DECL E6POS XP382={x 2180.9021,y 585.806824,z 1369.54504,a -78.3736267,b 58.1377296,c -93.7700119,s 6,t 27,e1 0.0,e2 0.0,e3 0.0,e4 0.0,e5 0.0,e6 0.0}
DECL FDAT FP382={TOOL_NO 1,BASE_NO 0,IPO_FRAME #BASE}
DECL PDAT PPDAT276={VEL 100.0,ACC 100.0,APO_DIST 100.0}
DECL E6POS XP383={x 1882.12,y 578.306091,z 982.650513,a -78.3796005,b 58.1366501,c -93.7758102,s 6,t 27,e1 0.0,e2 0.0,e3 0.0,e4 0.0,e5 0.0,e6 0.0}
DECL FDAT FP383={TOOL_NO 1,BASE_NO 0,IPO_FRAME #BASE}
DECL PDAT PPDAT277={VEL 100.0,ACC 100.0,APO_DIST 100.0}
DECL E6POS XP384={x 1882.09204,y 578.297729,z 939.258484,a -78.3842316,b 58.1358299,c -93.7813263,s 6,t 27,e1 0.0,e2 0.0,e3 0.0,e4 0.0,e5 0.0,e6 0.0}
DECL FDAT FP384={TOOL_NO 1,BASE_NO 0,IPO_FRAME #BASE}
DECL PDAT PPDAT278={VEL 100.0,ACC 100.0,APO_DIST 100.0}
DECL E6POS XP385={x 1882.10596,y 497.070801,z 1745.22595,a -88.2604828,b 58.8505211,c -105.352699,s 6,t 19,e1 0.0,e2 0.0,e3 0.0,e4 0.0,e5 0.0,e6 0.0}
DECL FDAT FP385={TOOL_NO 1,BASE_NO 0,IPO_FRAME #BASE}
DECL PDAT PPDAT279={VEL 100.0,ACC 100.0,APO_DIST 100.0}
DECL E6POS XP386={x 1882.10498,y 109.2248,z 1745.24194,a -43.191761,b 40.938839,c -48.9825897,s 6,t 19,e1 0.0,e2 0.0,e3 0.0,e4 0.0,e5 0.0,e6 0.0}
DECL FDAT FP386={TOOL_NO 1,BASE_NO 0,IPO_FRAME #BASE}
DECL PDAT PPDAT280={VEL 100.0,ACC 100.0,APO_DIST 100.0}
DECL E6POS XP387={x 1882.12097,y 109.308701,z 1745.27405,a 7.98916388,b -56.2097092,c 176.517807,s 6,t 27,e1 0.0,e2 0.0,e3 0.0,e4 0.0,e5 0.0,e6 0.0}
DECL FDAT FP387={TOOL_NO 1,BASE_NO 0,IPO_FRAME #BASE}
DECL PDAT PPDAT281={VEL 100.0,ACC 100.0,APO_DIST 100.0}
DECL E6POS XP388={x 1580.30603,y 109.311897,z 1338.53003,a 29.1239491,b -3.817909,c -177.125595,s 6,t 27,e1 0.0,e2 0.0,e3 0.0,e4 0.0,e5 0.0,e6 0.0}
DECL FDAT FP388={TOOL_NO 1,BASE_NO 0,IPO_FRAME #BASE}
DECL PDAT PPDAT282={VEL 100.0,ACC 100.0,APO_DIST 100.0}
DECL E6POS XP389={x 55.3110695,y 943.681396,z 1978.17395,a -6.70130014,b 52.5186882,c -94.4837189,s 2,t 11,e1 0.0,e2 0.0,e3 0.0,e4 0.0,e5 0.0,e6 0.0}
DECL FDAT FP389={TOOL_NO 1,BASE_NO 0,IPO_FRAME #BASE}
DECL PDAT PPDAT283={VEL 100.0,ACC 25.0,APO_DIST 100.0}
DECL E6POS XP390={x 1620.0,y 0.0,z 2195.0,a -90.0,b 59.9998817,c -90.0,s 2,t 2,e1 0.0,e2 0.0,e3 0.0,e4 0.0,e5 0.0,e6 0.0}
DECL FDAT FP390={TOOL_NO 1,BASE_NO 0,IPO_FRAME #BASE}
DECL PDAT PPDAT284={VEL 100.0,ACC 100.0,APO_DIST 100.0}
DECL E6POS XP391={x 1721.71704,y 98.0797729,z 1269.401,a -89.9984894,b 59.9988289,c -89.9980927,s 6,t 27,e1 0.0,e2 0.0,e3 0.0,e4 0.0,e5 0.0,e6 0.0}
DECL FDAT FP391={TOOL_NO 1,BASE_NO 0,IPO_FRAME #BASE}
DECL PDAT PPDAT285={VEL 100.0,ACC 100.0,APO_DIST 100.0}
DECL E6POS XP392={x 1730.89404,y 101.730797,z 1269.375,a -89.9981079,b 59.9989815,c -89.9963837,s 6,t 27,e1 0.0,e2 0.0,e3 0.0,e4 0.0,e5 0.0,e6 0.0}
DECL FDAT FP392={TOOL_NO 1,BASE_NO 0,IPO_FRAME #BASE}
DECL PDAT PPDAT286={VEL 100.0,ACC 100.0,APO_DIST 100.0}
DECL E6POS XP393={x 1730.89404,y 101.730797,z 1269.375,a -89.9981079,b 59.9989815,c -89.9963837,s 6,t 27,e1 0.0,e2 0.0,e3 0.0,e4 0.0,e5 0.0,e6 0.0}
DECL FDAT FP393={TOOL_NO 1,BASE_NO 0,IPO_FRAME #BASE}
DECL LDAT LCPDAT97={VEL 2.0,ACC 100.0,APO_DIST 100.0,APO_FAC 50.0}
DECL E6POS XP394={x 1730.89404,y 101.730797,z 1269.375,a -89.9981079,b 59.9989815,c -89.9963837,s 6,t 27,e1 0.0,e2 0.0,e3 0.0,e4 0.0,e5 0.0,e6 0.0}
DECL FDAT FP394={TOOL_NO 1,BASE_NO 0,IPO_FRAME #BASE}
DECL LDAT LCPDAT98={VEL 2.0,ACC 100.0,APO_DIST 100.0,APO_FAC 50.0}
DECL E6POS XP395={x 1721.30396,y 101.718201,z 1269.37402,a -89.9990005,b 59.9981804,c -89.9970932,s 6,t 27,e1 0.0,e2 0.0,e3 0.0,e4 0.0,e5 0.0,e6 0.0}
DECL FDAT FP395={TOOL_NO 1,BASE_NO 0,IPO_FRAME #BASE}
DECL LDAT LCPDAT99={VEL 2.0,ACC 100.0,APO_DIST 100.0,APO_FAC 50.0}
DECL E6POS XP396={x 1721.30896,y 95.7696762,z 1269.37903,a -89.9983902,b 59.9984283,c -89.9962692,s 6,t 27,e1 0.0,e2 0.0,e3 0.0,e4 0.0,e5 0.0,e6 0.0}
DECL FDAT FP396={TOOL_NO 1,BASE_NO 0,IPO_FRAME #BASE}
DECL LDAT LCPDAT100={VEL 2.0,ACC 100.0,APO_DIST 100.0,APO_FAC 50.0}
DECL E6POS XP397={x 1727.48706,y 95.7749023,z 1269.40405,a -89.994957,b 59.999321,c -89.9919434,s 6,t 27,e1 0.0,e2 0.0,e3 0.0,e4 0.0,e5 0.0,e6 0.0}
DECL FDAT FP397={TOOL_NO 1,BASE_NO 0,IPO_FRAME #BASE}
DECL LDAT LCPDAT101={VEL 2.0,ACC 100.0,APO_DIST 100.0,APO_FAC 50.0}
DECL E6POS XP398={x 1727.49194,y 99.8509369,z 1269.41504,a -89.9935379,b 60.0002289,c -89.9901505,s 6,t 27,e1 0.0,e2 0.0,e3 0.0,e4 0.0,e5 0.0,e6 0.0}
DECL FDAT FP398={TOOL_NO 1,BASE_NO 0,IPO_FRAME #BASE}
DECL LDAT LCPDAT102={VEL 2.0,ACC 100.0,APO_DIST 100.0,APO_FAC 50.0}
DECL E6POS XP399={x 1727.49194,y 99.8509369,z 1269.41504,a -89.9935379,b 60.0002289,c -89.9901505,s 6,t 27,e1 0.0,e2 0.0,e3 0.0,e4 0.0,e5 0.0,e6 0.0}
DECL FDAT FP399={TOOL_NO 1,BASE_NO 0,IPO_FRAME #BASE}
DECL PDAT PPDAT287={VEL 100.0,ACC 100.0,APO_DIST 100.0}
DECL E6POS XP400={x 1727.49805,y 9.73986816,z 1288.27502,a -89.9890137,b 68.490097,c -89.9850311,s 6,t 27,e1 0.0,e2 0.0,e3 0.0,e4 0.0,e5 0.0,e6 0.0}
DECL FDAT FP400={TOOL_NO 1,BASE_NO 0,IPO_FRAME #BASE}
DECL PDAT PPDAT288={VEL 100.0,ACC 100.0,APO_DIST 100.0}
DECL E6POS XP401={x 1825.16003,y 8.47059917,z 1266.86694,a -89.9738693,b 68.4893494,c -89.9686432,s 6,t 27,e1 0.0,e2 0.0,e3 0.0,e4 0.0,e5 0.0,e6 0.0}
DECL FDAT FP401={TOOL_NO 1,BASE_NO 0,IPO_FRAME #BASE}
DECL PDAT PPDAT289={VEL 100.0,ACC 100.0,APO_DIST 100.0}
DECL E6POS XP402={x 1825.16003,y 8.47059917,z 1266.86694,a -89.9738693,b 68.4893494,c -89.9686432,s 6,t 27,e1 0.0,e2 0.0,e3 0.0,e4 0.0,e5 0.0,e6 0.0}
DECL FDAT FP402={TOOL_NO 1,BASE_NO 0,IPO_FRAME #BASE}
DECL LDAT LCPDAT103={VEL 2.0,ACC 100.0,APO_DIST 100.0,APO_FAC 50.0}
DECL E6POS XP403={x 1795.98206,y 8.45187664,z 1267.44702,a -89.9924164,b 68.4888229,c -89.9880981,s 6,t 27,e1 0.0,e2 0.0,e3 0.0,e4 0.0,e5 0.0,e6 0.0}
DECL FDAT FP403={TOOL_NO 1,BASE_NO 0,IPO_FRAME #BASE}
DECL LDAT LCPDAT104={VEL 2.0,ACC 100.0,APO_DIST 100.0,APO_FAC 50.0}
DECL E6POS XP404={x 1762.83203,y 8.4597578,z 1218.80896,a -89.9986496,b 68.4880295,c -89.995163,s 6,t 27,e1 0.0,e2 0.0,e3 0.0,e4 0.0,e5 0.0,e6 0.0}
DECL FDAT FP404={TOOL_NO 1,BASE_NO 0,IPO_FRAME #BASE}
DECL LDAT LCPDAT105={VEL 2.0,ACC 100.0,APO_DIST 100.0,APO_FAC 50.0}
DECL E6POS XP405={x 1714.34094,y 9.04022121,z 1220.41504,a -90.0047531,b 68.486908,c -90.0016937,s 6,t 27,e1 0.0,e2 0.0,e3 0.0,e4 0.0,e5 0.0,e6 0.0}
DECL FDAT FP405={TOOL_NO 1,BASE_NO 0,IPO_FRAME #BASE}
DECL LDAT LCPDAT106={VEL 2.0,ACC 100.0,APO_DIST 100.0,APO_FAC 50.0}
DECL E6POS XP406={x 1787.46497,y 1.54117298,z 1305.14099,a -89.9851837,b 68.4879913,c -89.9798126,s 6,t 27,e1 0.0,e2 0.0,e3 0.0,e4 0.0,e5 0.0,e6 0.0}
DECL FDAT FP406={TOOL_NO 1,BASE_NO 0,IPO_FRAME #BASE}
DECL PDAT PPDAT290={VEL 100.0,ACC 100.0,APO_DIST 100.0}
DECL E6POS XP407={x 6.87235498,y -107.955902,z 3197.98999,a -95.3498535,b 3.01419806,c -0.477443188,s 2,t 10,e1 0.0,e2 0.0,e3 0.0,e4 0.0,e5 0.0,e6 0.0}
DECL FDAT FP407={TOOL_NO 1,BASE_NO 0,IPO_FRAME #BASE}
DECL PDAT PPDAT291={VEL 100.0,ACC 100.0,APO_DIST 100.0}
DECL E6POS XP408={x -2321.86401,y -437.479095,z 1523.60596,a -44.4752808,b -52.6538696,c 48.7558517,s 6,t 26,e1 0.0,e2 0.0,e3 0.0,e4 0.0,e5 0.0,e6 0.0}
DECL FDAT FP408={TOOL_NO 1,BASE_NO 0,IPO_FRAME #BASE}
DECL PDAT PPDAT292={VEL 100.0,ACC 100.0,APO_DIST 100.0}
DECL E6POS XP409={x 2083.62109,y -1113.97803,z 1523.60205,a 96.7235031,b -52.6538696,c 48.7562599,s 6,t 26,e1 0.0,e2 0.0,e3 0.0,e4 0.0,e5 0.0,e6 0.0}
DECL FDAT FP409={TOOL_NO 1,BASE_NO 0,IPO_FRAME #BASE}
DECL PDAT PPDAT293={VEL 100.0,ACC 100.0,APO_DIST 100.0}
DECL E6POS XP410={x 1843.23206,y -297.672211,z 1892.20703,a -104.636902,b 62.3937492,c -97.5844193,s 6,t 18,e1 0.0,e2 0.0,e3 0.0,e4 0.0,e5 0.0,e6 0.0}
DECL FDAT FP410={TOOL_NO 1,BASE_NO 0,IPO_FRAME #BASE}
DECL PDAT PPDAT294={VEL 100.0,ACC 100.0,APO_DIST 100.0}
DECL E6POS XP411={x 1891.35901,y -309.263092,z 920.833923,a -96.7764893,b 62.3960686,c -97.579422,s 6,t 18,e1 0.0,e2 0.0,e3 0.0,e4 0.0,e5 0.0,e6 0.0}
DECL FDAT FP411={TOOL_NO 1,BASE_NO 0,IPO_FRAME #BASE}
DECL PDAT PPDAT295={VEL 100.0,ACC 100.0,APO_DIST 100.0}
DECL E6POS XP412={x 1891.36206,y -309.26709,z 1131.79297,a -96.7787933,b 62.396759,c -97.5819702,s 6,t 18,e1 0.0,e2 0.0,e3 0.0,e4 0.0,e5 0.0,e6 0.0}
DECL FDAT FP412={TOOL_NO 1,BASE_NO 0,IPO_FRAME #BASE}
DECL PDAT PPDAT296={VEL 100.0,ACC 100.0,APO_DIST 100.0}
DECL E6POS XP413={x 1891.35803,y -150.701401,z 1131.78699,a -96.7800903,b 62.3966904,c -97.5833969,s 6,t 18,e1 0.0,e2 0.0,e3 0.0,e4 0.0,e5 0.0,e6 0.0}
DECL FDAT FP413={TOOL_NO 1,BASE_NO 0,IPO_FRAME #BASE}
DECL PDAT PPDAT297={VEL 100.0,ACC 100.0,APO_DIST 100.0}
DECL E6POS XP414={x 1891.39001,y -150.693405,z 1087.95801,a -96.7599106,b 62.3970795,c -97.5624237,s 6,t 18,e1 0.0,e2 0.0,e3 0.0,e4 0.0,e5 0.0,e6 0.0}
DECL FDAT FP414={TOOL_NO 1,BASE_NO 0,IPO_FRAME #BASE}
DECL PDAT PPDAT298={VEL 100.0,ACC 100.0,APO_DIST 100.0}
DECL E6POS XP415={x 1788.51697,y 1.54148304,z 1085.06396,a -89.9759216,b 68.4883728,c -89.9696884,s 6,t 27,e1 0.0,e2 0.0,e3 0.0,e4 0.0,e5 0.0,e6 0.0}
DECL FDAT FP415={TOOL_NO 1,BASE_NO 0,IPO_FRAME #BASE}
DECL PDAT PPDAT299={VEL 100.0,ACC 100.0,APO_DIST 100.0}
DECL E6POS XP416={x 1788.51697,y 1.54148304,z 1085.06396,a -89.9759216,b 68.4883728,c -89.9696884,s 6,t 27,e1 0.0,e2 0.0,e3 0.0,e4 0.0,e5 0.0,e6 0.0}
DECL FDAT FP416={TOOL_NO 1,BASE_NO 0,IPO_FRAME #BASE}
DECL LDAT LCPDAT107={VEL 2.0,ACC 100.0,APO_DIST 100.0,APO_FAC 50.0}
DECL E6POS XP417={x 1781.58704,y -240.441803,z 1083.771,a -89.9750977,b 68.4889297,c -89.9688263,s 6,t 18,e1 0.0,e2 0.0,e3 0.0,e4 0.0,e5 0.0,e6 0.0}
DECL FDAT FP417={TOOL_NO 1,BASE_NO 0,IPO_FRAME #BASE}
DECL LDAT LCPDAT108={VEL 2.0,ACC 100.0,APO_DIST 100.0,APO_FAC 50.0}
DECL E6POS XP418={x 1857.57495,y -189.287598,z 1190.64795,a -5.03419781,b 68.481781,c -89.9884262,s 6,t 50,e1 0.0,e2 0.0,e3 0.0,e4 0.0,e5 0.0,e6 0.0}
DECL FDAT FP418={TOOL_NO 1,BASE_NO 0,IPO_FRAME #BASE}
DECL PDAT PPDAT300={VEL 100.0,ACC 100.0,APO_DIST 100.0}
DECL E6POS XP419={x 1857.57104,y -189.290497,z 1089.01599,a -5.03386116,b 68.4827805,c -89.9877167,s 6,t 50,e1 0.0,e2 0.0,e3 0.0,e4 0.0,e5 0.0,e6 0.0}
DECL FDAT FP419={TOOL_NO 1,BASE_NO 0,IPO_FRAME #BASE}
DECL PDAT PPDAT301={VEL 100.0,ACC 100.0,APO_DIST 100.0}
DECL E6POS XP420={x 1857.57104,y -189.290497,z 1089.01599,a -5.03386116,b 68.4827805,c -89.9877167,s 6,t 50,e1 0.0,e2 0.0,e3 0.0,e4 0.0,e5 0.0,e6 0.0}
DECL FDAT FP420={TOOL_NO 1,BASE_NO 0,IPO_FRAME #BASE}
DECL LDAT LCPDAT109={VEL 2.0,ACC 100.0,APO_DIST 100.0,APO_FAC 50.0}
DECL E6POS XP421={x 2014.16101,y -191.725006,z 1089.02905,a -5.03730679,b 68.4811783,c -89.9894867,s 6,t 50,e1 0.0,e2 0.0,e3 0.0,e4 0.0,e5 0.0,e6 0.0}
DECL FDAT FP421={TOOL_NO 1,BASE_NO 0,IPO_FRAME #BASE}
DECL LDAT LCPDAT110={VEL 2.0,ACC 100.0,APO_DIST 100.0,APO_FAC 50.0}
DECL E6POS XP422={x 2014.16101,y -191.725006,z 1089.02905,a -5.03730679,b 68.4811783,c -89.9894867,s 6,t 50,e1 0.0,e2 0.0,e3 0.0,e4 0.0,e5 0.0,e6 0.0}
DECL FDAT FP422={TOOL_NO 1,BASE_NO 0,IPO_FRAME #BASE}
DECL PDAT PPDAT302={VEL 100.0,ACC 100.0,APO_DIST 100.0}
DECL E6POS XP423={x 1938.26904,y -244.236496,z 1088.59204,a -91.4427872,b 68.4859772,c -89.9945831,s 6,t 18,e1 0.0,e2 0.0,e3 0.0,e4 0.0,e5 0.0,e6 0.0}
DECL FDAT FP423={TOOL_NO 1,BASE_NO 0,IPO_FRAME #BASE}
DECL PDAT PPDAT303={VEL 100.0,ACC 100.0,APO_DIST 100.0}
DECL E6POS XP424={x 1938.27197,y -244.231201,z 1081.43005,a -91.440033,b 68.4871368,c -89.9929428,s 6,t 18,e1 0.0,e2 0.0,e3 0.0,e4 0.0,e5 0.0,e6 0.0}
DECL FDAT FP424={TOOL_NO 1,BASE_NO 0,IPO_FRAME #BASE}
DECL PDAT PPDAT304={VEL 100.0,ACC 100.0,APO_DIST 100.0}
DECL E6POS XP425={x 1938.27197,y -244.231201,z 1081.43005,a -91.440033,b 68.4871368,c -89.9929428,s 6,t 18,e1 0.0,e2 0.0,e3 0.0,e4 0.0,e5 0.0,e6 0.0}
DECL FDAT FP425={TOOL_NO 1,BASE_NO 0,IPO_FRAME #BASE}
DECL LDAT LCPDAT111={VEL 2.0,ACC 100.0,APO_DIST 100.0,APO_FAC 50.0}
DECL E6POS XP426={x 1951.03503,y 280.272705,z 1084.44604,a -91.4313889,b 68.4940109,c -89.9844894,s 6,t 27,e1 0.0,e2 0.0,e3 0.0,e4 0.0,e5 0.0,e6 0.0}
DECL FDAT FP426={TOOL_NO 1,BASE_NO 0,IPO_FRAME #BASE}
DECL LDAT LCPDAT112={VEL 2.0,ACC 100.0,APO_DIST 100.0,APO_FAC 50.0}
DECL E6POS XP427={x 1951.03503,y 280.272705,z 1084.44604,a -91.4313889,b 68.4940109,c -89.9844894,s 6,t 27,e1 0.0,e2 0.0,e3 0.0,e4 0.0,e5 0.0,e6 0.0}
DECL FDAT FP427={TOOL_NO 1,BASE_NO 0,IPO_FRAME #BASE}
DECL PDAT PPDAT305={VEL 100.0,ACC 100.0,APO_DIST 100.0}
DECL E6POS XP428={x 2026.85901,y 334.200104,z 1105.98096,a -4.45665598,b 68.4910431,c -89.9797287,s 6,t 51,e1 0.0,e2 0.0,e3 0.0,e4 0.0,e5 0.0,e6 0.0}
DECL FDAT FP428={TOOL_NO 1,BASE_NO 0,IPO_FRAME #BASE}
DECL PDAT PPDAT306={VEL 100.0,ACC 100.0,APO_DIST 100.0}
DECL E6POS XP429={x 2026.85596,y 334.200012,z 1089.23096,a -4.45706797,b 68.4920731,c -89.9801331,s 6,t 51,e1 0.0,e2 0.0,e3 0.0,e4 0.0,e5 0.0,e6 0.0}
DECL FDAT FP429={TOOL_NO 1,BASE_NO 0,IPO_FRAME #BASE}
DECL LDAT LCPDAT113={VEL 2.0,ACC 100.0,APO_DIST 100.0,APO_FAC 50.0}
DECL E6POS XP430={x 2026.85596,y 334.200012,z 1089.23096,a -4.45706797,b 68.4920731,c -89.9801331,s 6,t 51,e1 0.0,e2 0.0,e3 0.0,e4 0.0,e5 0.0,e6 0.0}
DECL FDAT FP430={TOOL_NO 1,BASE_NO 0,IPO_FRAME #BASE}
DECL LDAT LCPDAT114={VEL 2.0,ACC 100.0,APO_DIST 100.0,APO_FAC 50.0}
DECL E6POS XP431={x 1867.99402,y 335.831604,z 1091.06995,a -4.45940113,b 68.4928665,c -89.9819336,s 6,t 51,e1 0.0,e2 0.0,e3 0.0,e4 0.0,e5 0.0,e6 0.0}
DECL FDAT FP431={TOOL_NO 1,BASE_NO 0,IPO_FRAME #BASE}
DECL LDAT LCPDAT115={VEL 2.0,ACC 100.0,APO_DIST 100.0,APO_FAC 50.0}
DECL E6POS XP432={x 1867.99402,y 335.831604,z 1091.06995,a -4.45940113,b 68.4928665,c -89.9819336,s 6,t 51,e1 0.0,e2 0.0,e3 0.0,e4 0.0,e5 0.0,e6 0.0}
DECL FDAT FP432={TOOL_NO 1,BASE_NO 0,IPO_FRAME #BASE}
DECL PDAT PPDAT307={VEL 100.0,ACC 100.0,APO_DIST 100.0}
DECL E6POS XP433={x 1801.823,y 283.612,z 1101.84595,a -95.9969177,b 68.3930435,c -93.1611633,s 6,t 27,e1 0.0,e2 0.0,e3 0.0,e4 0.0,e5 0.0,e6 0.0}
DECL FDAT FP433={TOOL_NO 1,BASE_NO 0,IPO_FRAME #BASE}
DECL PDAT PPDAT308={VEL 100.0,ACC 100.0,APO_DIST 100.0}
DECL E6POS XP434={x 1801.83801,y 283.613007,z 1086.224,a -95.9930725,b 68.3924332,c -93.1558304,s 6,t 27,e1 0.0,e2 0.0,e3 0.0,e4 0.0,e5 0.0,e6 0.0}
DECL FDAT FP434={TOOL_NO 1,BASE_NO 0,IPO_FRAME #BASE}
DECL PDAT PPDAT309={VEL 100.0,ACC 100.0,APO_DIST 100.0}
DECL E6POS XP435={x 1801.84705,y 284.174896,z 1086.23096,a -95.9924088,b 68.3929901,c -93.1550217,s 6,t 27,e1 0.0,e2 0.0,e3 0.0,e4 0.0,e5 0.0,e6 0.0}
DECL FDAT FP435={TOOL_NO 1,BASE_NO 0,IPO_FRAME #BASE}
DECL LDAT LCPDAT116={VEL 2.0,ACC 100.0,APO_DIST 100.0,APO_FAC 50.0}
DECL E6POS XP436={x 1800.22595,y 216.311996,z 1086.229,a -95.9936371,b 68.3931732,c -93.155899,s 6,t 27,e1 0.0,e2 0.0,e3 0.0,e4 0.0,e5 0.0,e6 0.0}
DECL FDAT FP436={TOOL_NO 1,BASE_NO 0,IPO_FRAME #BASE}
DECL LDAT LCPDAT117={VEL 2.0,ACC 100.0,APO_DIST 100.0,APO_FAC 50.0}
DECL E6POS XP437={x 1800.22205,y 198.541901,z 1134.521,a -95.9973221,b 68.3924637,c -93.1600571,s 6,t 27,e1 0.0,e2 0.0,e3 0.0,e4 0.0,e5 0.0,e6 0.0}
DECL E6POS XP438={x 1800.23499,y 178.785706,z 1109.75195,a -95.9939728,b 68.3902435,c -93.1574936,s 6,t 27,e1 0.0,e2 0.0,e3 0.0,e4 0.0,e5 0.0,e6 0.0}
DECL FDAT FP438={TOOL_NO 1,BASE_NO 0,IPO_FRAME #BASE}
DECL LDAT LCPDAT118={VEL 2.0,ACC 100.0,APO_DIST 100.0,APO_FAC 50.0}
DECL E6POS XP439={x 1800.23596,y 178.768494,z 1086.354,a -95.9938278,b 68.3870468,c -93.1533966,s 6,t 27,e1 0.0,e2 0.0,e3 0.0,e4 0.0,e5 0.0,e6 0.0}
DECL FDAT FP439={TOOL_NO 1,BASE_NO 0,IPO_FRAME #BASE}
DECL LDAT LCPDAT119={VEL 2.0,ACC 100.0,APO_DIST 100.0,APO_FAC 50.0}
DECL E6POS XP440={x 1797.48499,y 99.9996567,z 1086.354,a -95.9934998,b 68.3869934,c -93.1527481,s 6,t 27,e1 0.0,e2 0.0,e3 0.0,e4 0.0,e5 0.0,e6 0.0}
DECL FDAT FP440={TOOL_NO 1,BASE_NO 0,IPO_FRAME #BASE}
DECL LDAT LCPDAT120={VEL 2.0,ACC 100.0,APO_DIST 100.0,APO_FAC 50.0}
DECL E6POS XP441={x 1708.21704,y 230.690506,z 1194.828,a -77.1536865,b 58.7134018,c -71.4141769,s 6,t 27,e1 0.0,e2 0.0,e3 0.0,e4 0.0,e5 0.0,e6 0.0}
DECL FDAT FP441={TOOL_NO 1,BASE_NO 0,IPO_FRAME #BASE}
DECL PDAT PPDAT310={VEL 100.0,ACC 100.0,APO_DIST 100.0}
DECL E6POS XP442={x 1709.53699,y 242.714905,z 1080.94397,a -77.1506729,b 58.7134705,c -71.4099426,s 6,t 27,e1 0.0,e2 0.0,e3 0.0,e4 0.0,e5 0.0,e6 0.0}
DECL FDAT FP442={TOOL_NO 1,BASE_NO 0,IPO_FRAME #BASE}
DECL PDAT PPDAT311={VEL 100.0,ACC 100.0,APO_DIST 100.0}
DECL E6POS XP443={x 1709.53699,y 242.714905,z 1080.94397,a -77.1506729,b 58.7134705,c -71.4099426,s 6,t 27,e1 0.0,e2 0.0,e3 0.0,e4 0.0,e5 0.0,e6 0.0}
DECL FDAT FP443={TOOL_NO 1,BASE_NO 0,IPO_FRAME #BASE}
DECL LDAT LCPDAT121={VEL 2.0,ACC 100.0,APO_DIST 100.0,APO_FAC 50.0}
DECL E6POS XP444={x 1706.01196,y 92.4064713,z 1079.61096,a -77.1516113,b 58.7126198,c -71.4103317,s 6,t 27,e1 0.0,e2 0.0,e3 0.0,e4 0.0,e5 0.0,e6 0.0}
DECL FDAT FP444={TOOL_NO 1,BASE_NO 0,IPO_FRAME #BASE}
DECL LDAT LCPDAT122={VEL 2.0,ACC 100.0,APO_DIST 100.0,APO_FAC 50.0}
DECL E6POS XP445={x 1706.01099,y 92.4069672,z 1289.64502,a -77.1514664,b 58.712719,c -71.4103165,s 6,t 27,e1 0.0,e2 0.0,e3 0.0,e4 0.0,e5 0.0,e6 0.0}
DECL FDAT FP445={TOOL_NO 1,BASE_NO 0,IPO_FRAME #BASE}
DECL PDAT PPDAT312={VEL 100.0,ACC 100.0,APO_DIST 100.0}
DECL E6POS XP446={x 1625.10095,y -190.573196,z 915.192627,a -77.1490631,b 58.7168884,c -71.4077988,s 6,t 18,e1 0.0,e2 0.0,e3 0.0,e4 0.0,e5 0.0,e6 0.0}
DECL FDAT FP446={TOOL_NO 1,BASE_NO 0,IPO_FRAME #BASE}
DECL PDAT PPDAT313={VEL 100.0,ACC 100.0,APO_DIST 100.0}
DECL E6POS XP447={x 1625.10095,y -190.573196,z 915.192627,a -77.1490631,b 58.7168884,c -71.4077988,s 6,t 18,e1 0.0,e2 0.0,e3 0.0,e4 0.0,e5 0.0,e6 0.0}
DECL FDAT FP447={TOOL_NO 1,BASE_NO 0,IPO_FRAME #BASE}
DECL LDAT LCPDAT123={VEL 2.0,ACC 100.0,APO_DIST 100.0,APO_FAC 50.0}
DECL E6POS XP448={x 1620.70203,y -356.353699,z 913.115417,a -77.1501923,b 58.7190208,c -71.4090805,s 6,t 18,e1 0.0,e2 0.0,e3 0.0,e4 0.0,e5 0.0,e6 0.0}
DECL FDAT FP448={TOOL_NO 1,BASE_NO 0,IPO_FRAME #BASE}
DECL LDAT LCPDAT124={VEL 2.0,ACC 100.0,APO_DIST 100.0,APO_FAC 50.0}
DECL E6POS XP449={x 1626.60706,y -375.643707,z 913.122986,a -77.1490707,b 58.7185707,c -71.40802,s 6,t 18,e1 0.0,e2 0.0,e3 0.0,e4 0.0,e5 0.0,e6 0.0}
DECL E6POS XP450={x 1651.60303,y -391.266998,z 912.728394,a -77.1474991,b 58.717701,c -71.4053802,s 6,t 18,e1 0.0,e2 0.0,e3 0.0,e4 0.0,e5 0.0,e6 0.0}
DECL FDAT FP450={TOOL_NO 1,BASE_NO 0,IPO_FRAME #BASE}
DECL LDAT LCPDAT125={VEL 2.0,ACC 100.0,APO_DIST 100.0,APO_FAC 50.0}
DECL E6POS XP451={x 1651.60303,y -391.266998,z 912.728394,a -77.1474991,b 58.717701,c -71.4053802,s 6,t 18,e1 0.0,e2 0.0,e3 0.0,e4 0.0,e5 0.0,e6 0.0}
DECL FDAT FP451={TOOL_NO 1,BASE_NO 0,IPO_FRAME #BASE}
DECL LDAT LCPDAT126={VEL 2.0,ACC 100.0,APO_DIST 100.0,APO_FAC 50.0}
DECL E6POS XP452={x 1877.198,y -398.11499,z 910.503418,a -77.1458435,b 58.7178192,c -71.4037476,s 6,t 18,e1 0.0,e2 0.0,e3 0.0,e4 0.0,e5 0.0,e6 0.0}
DECL FDAT FP452={TOOL_NO 1,BASE_NO 0,IPO_FRAME #BASE}
DECL LDAT LCPDAT127={VEL 2.0,ACC 100.0,APO_DIST 100.0,APO_FAC 50.0}
DECL E6POS XP453={x 1902.11096,y -390.78891,z 910.030579,a -77.1470032,b 58.7169991,c -71.404808,s 6,t 18,e1 0.0,e2 0.0,e3 0.0,e4 0.0,e5 0.0,e6 0.0}
DECL E6POS XP454={x 1917.34802,y -364.729797,z 908.523926,a -77.1485367,b 58.7078781,c -71.4084473,s 6,t 18,e1 0.0,e2 0.0,e3 0.0,e4 0.0,e5 0.0,e6 0.0}
DECL FDAT FP454={TOOL_NO 1,BASE_NO 0,IPO_FRAME #BASE}
DECL LDAT LCPDAT128={VEL 2.0,ACC 100.0,APO_DIST 100.0,APO_FAC 50.0}
DECL E6POS XP455={x 1917.34802,y -364.729797,z 908.523926,a -77.1485367,b 58.7078781,c -71.4084473,s 6,t 18,e1 0.0,e2 0.0,e3 0.0,e4 0.0,e5 0.0,e6 0.0}
DECL FDAT FP455={TOOL_NO 1,BASE_NO 0,IPO_FRAME #BASE}
DECL LDAT LCPDAT129={VEL 2.0,ACC 100.0,APO_DIST 100.0,APO_FAC 50.0}
DECL E6POS XP456={x 1921.93506,y -200.479202,z 909.75769,a -77.1460266,b 58.7062302,c -71.4055176,s 6,t 18,e1 0.0,e2 0.0,e3 0.0,e4 0.0,e5 0.0,e6 0.0}
DECL FDAT FP456={TOOL_NO 1,BASE_NO 0,IPO_FRAME #BASE}
DECL LDAT LCPDAT130={VEL 2.0,ACC 100.0,APO_DIST 100.0,APO_FAC 50.0}
DECL E6POS XP457={x 1904.64905,y -200.408203,z 909.721985,a -77.1480331,b 58.7104607,c -71.4070206,s 6,t 18,e1 0.0,e2 0.0,e3 0.0,e4 0.0,e5 0.0,e6 0.0}
DECL FDAT FP457={TOOL_NO 1,BASE_NO 0,IPO_FRAME #BASE}
DECL LDAT LCPDAT131={VEL 2.0,ACC 100.0,APO_DIST 100.0,APO_FAC 50.0}
DECL E6POS XP458={x 1904.64905,y -200.408203,z 909.721985,a -77.1480331,b 58.7104607,c -71.4070206,s 6,t 18,e1 0.0,e2 0.0,e3 0.0,e4 0.0,e5 0.0,e6 0.0}
DECL FDAT FP458={TOOL_NO 1,BASE_NO 0,IPO_FRAME #BASE}
DECL PDAT PPDAT314={VEL 100.0,ACC 100.0,APO_DIST 100.0}
DECL E6POS XP459={x 1445.38599,y -160.803207,z 1290.83801,a 25.9863892,b 41.1141396,c -156.642197,s 6,t 18,e1 0.0,e2 0.0,e3 0.0,e4 0.0,e5 0.0,e6 0.0}
DECL FDAT FP459={TOOL_NO 1,BASE_NO 0,IPO_FRAME #BASE}
DECL PDAT PPDAT315={VEL 100.0,ACC 100.0,APO_DIST 100.0}
DECL E6POS XP460={x 1248.83606,y -271.152313,z 804.615112,a 25.9864807,b 41.1133118,c -156.642197,s 6,t 18,e1 0.0,e2 0.0,e3 0.0,e4 0.0,e5 0.0,e6 0.0}
DECL FDAT FP460={TOOL_NO 1,BASE_NO 0,IPO_FRAME #BASE}
DECL PDAT PPDAT316={VEL 100.0,ACC 100.0,APO_DIST 100.0}
DECL E6POS XP461={x 1327.15002,y -77.0415573,z 314.4617,a 25.98666,b 41.113369,c -156.641693,s 6,t 18,e1 0.0,e2 0.0,e3 0.0,e4 0.0,e5 0.0,e6 0.0}
DECL FDAT FP461={TOOL_NO 1,BASE_NO 0,IPO_FRAME #BASE}
DECL PDAT PPDAT317={VEL 100.0,ACC 100.0,APO_DIST 100.0}
DECL E6POS XP462={x 1327.15002,y -77.0415573,z 314.4617,a 25.98666,b 41.113369,c -156.641693,s 6,t 18,e1 0.0,e2 0.0,e3 0.0,e4 0.0,e5 0.0,e6 0.0}
DECL FDAT FP462={TOOL_NO 1,BASE_NO 0,IPO_FRAME #BASE}
DECL LDAT LCPDAT132={VEL 2.0,ACC 100.0,APO_DIST 100.0,APO_FAC 50.0}
DECL E6POS XP463={x 1325.04602,y -119.980499,z 314.466003,a 25.9877205,b 41.1126709,c -156.641495,s 6,t 18,e1 0.0,e2 0.0,e3 0.0,e4 0.0,e5 0.0,e6 0.0}
DECL FDAT FP463={TOOL_NO 1,BASE_NO 0,IPO_FRAME #BASE}
DECL LDAT LCPDAT133={VEL 2.0,ACC 100.0,APO_DIST 100.0,APO_FAC 50.0}
DECL E6POS XP464={x 1325.04602,y -119.980499,z 314.466003,a 25.9877205,b 41.1126709,c -156.641495,s 6,t 18,e1 0.0,e2 0.0,e3 0.0,e4 0.0,e5 0.0,e6 0.0}
DECL FDAT FP464={TOOL_NO 1,BASE_NO 0,IPO_FRAME #BASE}
DECL PDAT PPDAT318={VEL 100.0,ACC 100.0,APO_DIST 100.0}
DECL E6POS XP465={x 1273.81201,y -137.484802,z 340.795685,a 61.2980118,b 9.6628418,c -154.180496,s 6,t 18,e1 0.0,e2 0.0,e3 0.0,e4 0.0,e5 0.0,e6 0.0}
DECL FDAT FP465={TOOL_NO 1,BASE_NO 0,IPO_FRAME #BASE}
DECL PDAT PPDAT319={VEL 100.0,ACC 100.0,APO_DIST 100.0}
DECL E6POS XP466={x 1537.71497,y -668.202698,z 171.415695,a 104.630501,b 11.8383102,c -163.363495,s 6,t 18,e1 0.0,e2 0.0,e3 0.0,e4 0.0,e5 0.0,e6 0.0}
DECL FDAT FP466={TOOL_NO 1,BASE_NO 0,IPO_FRAME #BASE}
DECL PDAT PPDAT320={VEL 100.0,ACC 100.0,APO_DIST 100.0}
DECL E6POS XP467={x 1562.52502,y -647.870789,z 113.460503,a 104.636703,b 11.8369703,c -163.356903,s 6,t 18,e1 0.0,e2 0.0,e3 0.0,e4 0.0,e5 0.0,e6 0.0}
DECL FDAT FP467={TOOL_NO 1,BASE_NO 0,IPO_FRAME #BASE}
DECL PDAT PPDAT321={VEL 100.0,ACC 100.0,APO_DIST 100.0}
DECL E6POS XP468={x 1562.52502,y -647.870789,z 113.460503,a 104.636703,b 11.8369703,c -163.356903,s 6,t 18,e1 0.0,e2 0.0,e3 0.0,e4 0.0,e5 0.0,e6 0.0}
DECL FDAT FP468={TOOL_NO 1,BASE_NO 0,IPO_FRAME #BASE}
DECL LDAT LCPDAT134={VEL 2.0,ACC 100.0,APO_DIST 100.0,APO_FAC 50.0}
DECL E6POS XP469={x 1650.46301,y -764.261719,z 141.7388,a 111.916603,b 12.6148796,c -162.760406,s 6,t 18,e1 0.0,e2 0.0,e3 0.0,e4 0.0,e5 0.0,e6 0.0}
DECL FDAT FP469={TOOL_NO 1,BASE_NO 0,IPO_FRAME #BASE}
DECL PDAT PPDAT322={VEL 100.0,ACC 100.0,APO_DIST 100.0}
DECL E6POS XP470={x 1736.82703,y -723.896973,z 128.705505,a 120.375099,b 11.2741404,c 178.413696,s 6,t 18,e1 0.0,e2 0.0,e3 0.0,e4 0.0,e5 0.0,e6 0.0}
DECL FDAT FP470={TOOL_NO 1,BASE_NO 0,IPO_FRAME #BASE}
DECL PDAT PPDAT323={VEL 100.0,ACC 100.0,APO_DIST 100.0}
DECL E6POS XP471={x 1688.82605,y -677.752686,z 41.5209808,a 120.434601,b 11.2534103,c 178.413101,s 6,t 18,e1 0.0,e2 0.0,e3 0.0,e4 0.0,e5 0.0,e6 0.0}
DECL FDAT FP471={TOOL_NO 1,BASE_NO 0,IPO_FRAME #BASE}
DECL PDAT PPDAT324={VEL 100.0,ACC 100.0,APO_DIST 100.0}
DECL E6POS XP472={x 1688.82605,y -677.752686,z 41.5209808,a 120.434601,b 11.2534103,c 178.413101,s 6,t 18,e1 0.0,e2 0.0,e3 0.0,e4 0.0,e5 0.0,e6 0.0}
DECL FDAT FP472={TOOL_NO 1,BASE_NO 0,IPO_FRAME #BASE}
DECL LDAT LCPDAT135={VEL 2.0,ACC 100.0,APO_DIST 100.0,APO_FAC 50.0}
DECL E6POS XP473={x 2098.49512,y -702.313293,z 25.9236202,a 120.298401,b 11.2801504,c 178.387405,s 6,t 16,e1 0.0,e2 0.0,e3 0.0,e4 0.0,e5 0.0,e6 0.0}
DECL FDAT FP473={TOOL_NO 1,BASE_NO 0,IPO_FRAME #BASE}
DECL LDAT LCPDAT136={VEL 2.0,ACC 100.0,APO_DIST 100.0,APO_FAC 50.0}
DECL E6POS XP474={x 2098.48389,y -702.309814,z 55.3821487,a 120.297897,b 11.2795696,c 178.387802,s 6,t 18,e1 0.0,e2 0.0,e3 0.0,e4 0.0,e5 0.0,e6 0.0}
DECL FDAT FP474={TOOL_NO 1,BASE_NO 0,IPO_FRAME #BASE}
DECL LDAT LCPDAT137={VEL 2.0,ACC 100.0,APO_DIST 100.0,APO_FAC 50.0}
DECL E6POS XP475={x 2115.11304,y -702.729614,z 55.6279488,a 120.275398,b 11.2933197,c 178.377502,s 6,t 16,e1 0.0,e2 0.0,e3 0.0,e4 0.0,e5 0.0,e6 0.0}
DECL FDAT FP475={TOOL_NO 1,BASE_NO 0,IPO_FRAME #BASE}
DECL LDAT LCPDAT138={VEL 2.0,ACC 100.0,APO_DIST 100.0,APO_FAC 50.0}
DECL E6POS XP476={x 2124.01392,y -702.980286,z 77.9356689,a 120.264397,b 11.3027401,c 178.372101,s 6,t 18,e1 0.0,e2 0.0,e3 0.0,e4 0.0,e5 0.0,e6 0.0}
DECL FDAT FP476={TOOL_NO 1,BASE_NO 0,IPO_FRAME #BASE}
DECL LDAT LCPDAT139={VEL 2.0,ACC 100.0,APO_DIST 100.0,APO_FAC 50.0}
DECL E6POS XP477={x 2124.03589,y -704.693481,z 434.082092,a 120.264,b 11.3042898,c 178.371002,s 6,t 18,e1 0.0,e2 0.0,e3 0.0,e4 0.0,e5 0.0,e6 0.0}
DECL FDAT FP477={TOOL_NO 1,BASE_NO 0,IPO_FRAME #BASE}
DECL LDAT LCPDAT140={VEL 2.0,ACC 100.0,APO_DIST 100.0,APO_FAC 50.0}
DECL E6POS XP478={x 1990.90906,y -701.373108,z 433.983612,a 120.269699,b 11.2985401,c 178.375702,s 6,t 18,e1 0.0,e2 0.0,e3 0.0,e4 0.0,e5 0.0,e6 0.0}
DECL FDAT FP478={TOOL_NO 1,BASE_NO 0,IPO_FRAME #BASE}
DECL LDAT LCPDAT141={VEL 2.0,ACC 100.0,APO_DIST 100.0,APO_FAC 50.0}
DECL E6POS XP479={x 1988.927,y -699.174316,z 60.8071785,a 120.2696,b 11.2961302,c 178.377594,s 6,t 18,e1 0.0,e2 0.0,e3 0.0,e4 0.0,e5 0.0,e6 0.0}
DECL FDAT FP479={TOOL_NO 1,BASE_NO 0,IPO_FRAME #BASE}
DECL LDAT LCPDAT142={VEL 2.0,ACC 100.0,APO_DIST 100.0,APO_FAC 50.0}
DECL E6POS XP480={x 2115.64795,y -703.102112,z 57.7487602,a 120.233398,b 11.3163996,c 178.362,s 6,t 16,e1 0.0,e2 0.0,e3 0.0,e4 0.0,e5 0.0,e6 0.0}
DECL FDAT FP480={TOOL_NO 1,BASE_NO 0,IPO_FRAME #BASE}
DECL LDAT LCPDAT143={VEL 2.0,ACC 100.0,APO_DIST 100.0,APO_FAC 50.0}
DECL E6POS XP481={x 2115.64795,y -703.102112,z 57.7487602,a 120.233398,b 11.3163996,c 178.362,s 6,t 16,e1 0.0,e2 0.0,e3 0.0,e4 0.0,e5 0.0,e6 0.0}
DECL FDAT FP481={TOOL_NO 1,BASE_NO 0,IPO_FRAME #BASE}
DECL PDAT PPDAT325={VEL 100.0,ACC 100.0,APO_DIST 100.0}
DECL E6POS XP482={x 2223.93091,y -790.63208,z 523.430725,a -163.255295,b 28.3873997,c -160.907394,s 6,t 18,e1 0.0,e2 0.0,e3 0.0,e4 0.0,e5 0.0,e6 0.0}
DECL FDAT FP482={TOOL_NO 1,BASE_NO 0,IPO_FRAME #BASE}
DECL PDAT PPDAT326={VEL 100.0,ACC 100.0,APO_DIST 100.0}
DECL E6POS XP483={x 2208.95093,y -745.331909,z 478.839996,a -166.892593,b 23.05056,c -174.636505,s 6,t 18,e1 0.0,e2 0.0,e3 0.0,e4 0.0,e5 0.0,e6 0.0}
DECL FDAT FP483={TOOL_NO 1,BASE_NO 0,IPO_FRAME #BASE}
DECL PDAT PPDAT327={VEL 100.0,ACC 100.0,APO_DIST 100.0}
DECL E6POS XP484={x 2480.60303,y -360.321411,z 663.894226,a -162.0504,b 40.5198593,c -168.634903,s 6,t 18,e1 0.0,e2 0.0,e3 0.0,e4 0.0,e5 0.0,e6 0.0}
DECL FDAT FP484={TOOL_NO 1,BASE_NO 0,IPO_FRAME #BASE}
DECL PDAT PPDAT328={VEL 100.0,ACC 100.0,APO_DIST 100.0}
DECL E6POS XP485={x 2481.25293,y -329.930511,z 671.163208,a -162.048096,b 40.5211296,c -168.631805,s 6,t 18,e1 0.0,e2 0.0,e3 0.0,e4 0.0,e5 0.0,e6 0.0}
DECL FDAT FP485={TOOL_NO 1,BASE_NO 0,IPO_FRAME #BASE}
DECL PDAT PPDAT329={VEL 100.0,ACC 100.0,APO_DIST 100.0}
DECL E6POS XP486={x 2481.25293,y -329.930511,z 671.163208,a -162.048096,b 40.5211296,c -168.631805,s 6,t 18,e1 0.0,e2 0.0,e3 0.0,e4 0.0,e5 0.0,e6 0.0}
DECL FDAT FP486={TOOL_NO 1,BASE_NO 0,IPO_FRAME #BASE}
DECL LDAT LCPDAT144={VEL 2.0,ACC 100.0,APO_DIST 100.0,APO_FAC 50.0}
DECL E6POS XP487={x 2477.89893,y -329.7995,z 318.438995,a -162.051498,b 40.5162697,c -168.640396,s 6,t 18,e1 0.0,e2 0.0,e3 0.0,e4 0.0,e5 0.0,e6 0.0}
DECL FDAT FP487={TOOL_NO 1,BASE_NO 0,IPO_FRAME #BASE}
DECL LDAT LCPDAT145={VEL 2.0,ACC 100.0,APO_DIST 100.0,APO_FAC 50.0}
DECL E6POS XP488={x 2477.89893,y -329.7995,z 318.438995,a -162.051498,b 40.5162697,c -168.640396,s 6,t 18,e1 0.0,e2 0.0,e3 0.0,e4 0.0,e5 0.0,e6 0.0}
DECL FDAT FP488={TOOL_NO 1,BASE_NO 0,IPO_FRAME #BASE}
DECL PDAT PPDAT330={VEL 100.0,ACC 100.0,APO_DIST 100.0}
DECL E6POS XP489={x 2516.39111,y -188.610901,z 627.18042,a -162.045502,b 40.5088196,c -168.629395,s 6,t 18,e1 0.0,e2 0.0,e3 0.0,e4 0.0,e5 0.0,e6 0.0}
DECL FDAT FP489={TOOL_NO 1,BASE_NO 0,IPO_FRAME #BASE}
DECL PDAT PPDAT331={VEL 100.0,ACC 100.0,APO_DIST 100.0}
DECL E6POS XP490={x 2494.11108,y -188.337494,z 627.181213,a -162.059906,b 40.500721,c -168.647507,s 6,t 18,e1 0.0,e2 0.0,e3 0.0,e4 0.0,e5 0.0,e6 0.0}
DECL FDAT FP490={TOOL_NO 1,BASE_NO 0,IPO_FRAME #BASE}
DECL PDAT PPDAT332={VEL 100.0,ACC 100.0,APO_DIST 100.0}
DECL E6POS XP491={x 2494.11108,y -188.337494,z 627.181213,a -162.059906,b 40.500721,c -168.647507,s 6,t 18,e1 0.0,e2 0.0,e3 0.0,e4 0.0,e5 0.0,e6 0.0}
DECL FDAT FP491={TOOL_NO 1,BASE_NO 0,IPO_FRAME #BASE}
DECL LDAT LCPDAT146={VEL 2.0,ACC 100.0,APO_DIST 100.0,APO_FAC 50.0}
DECL E6POS XP492={x 2490.08911,y -302.415009,z 625.75061,a -162.063004,b 40.4979286,c -168.653,s 6,t 18,e1 0.0,e2 0.0,e3 0.0,e4 0.0,e5 0.0,e6 0.0}
DECL FDAT FP492={TOOL_NO 1,BASE_NO 0,IPO_FRAME #BASE}
DECL LDAT LCPDAT147={VEL 2.0,ACC 100.0,APO_DIST 100.0,APO_FAC 50.0}
DECL E6POS XP493={x 2490.08594,y -302.415009,z 527.262817,a -162.062302,b 40.4976501,c -168.652496,s 6,t 18,e1 0.0,e2 0.0,e3 0.0,e4 0.0,e5 0.0,e6 0.0}
DECL FDAT FP493={TOOL_NO 1,BASE_NO 0,IPO_FRAME #BASE}
DECL LDAT LCPDAT148={VEL 2.0,ACC 100.0,APO_DIST 100.0,APO_FAC 50.0}
DECL E6POS XP494={x 2490.09204,y -187.837799,z 527.275879,a -162.062302,b 40.4984016,c -168.6521,s 6,t 18,e1 0.0,e2 0.0,e3 0.0,e4 0.0,e5 0.0,e6 0.0}
DECL FDAT FP494={TOOL_NO 1,BASE_NO 0,IPO_FRAME #BASE}
DECL LDAT LCPDAT149={VEL 2.0,ACC 100.0,APO_DIST 100.0,APO_FAC 50.0}
DECL E6POS XP495={x 2491.1499,y -187.852005,z 626.662781,a -162.061798,b 40.5001411,c -168.651001,s 6,t 18,e1 0.0,e2 0.0,e3 0.0,e4 0.0,e5 0.0,e6 0.0}
DECL FDAT FP495={TOOL_NO 1,BASE_NO 0,IPO_FRAME #BASE}
DECL LDAT LCPDAT150={VEL 2.0,ACC 100.0,APO_DIST 100.0,APO_FAC 50.0}
DECL E6POS XP496={x 2491.1499,y -187.852005,z 626.662781,a -162.061798,b 40.5001411,c -168.651001,s 6,t 18,e1 0.0,e2 0.0,e3 0.0,e4 0.0,e5 0.0,e6 0.0}
DECL FDAT FP496={TOOL_NO 1,BASE_NO 0,IPO_FRAME #BASE}
DECL PDAT PPDAT333={VEL 100.0,ACC 100.0,APO_DIST 100.0}
DECL E6POS XP497={x 2535.96509,y 231.158096,z 444.117096,a -162.057205,b 40.5109787,c -168.650497,s 6,t 19,e1 0.0,e2 0.0,e3 0.0,e4 0.0,e5 0.0,e6 0.0}
DECL FDAT FP497={TOOL_NO 1,BASE_NO 0,IPO_FRAME #BASE}
DECL PDAT PPDAT334={VEL 100.0,ACC 100.0,APO_DIST 100.0}
DECL E6POS XP498={x 2502.83008,y 203.052399,z 526.657227,a -162.090805,b 40.4880486,c -168.669601,s 6,t 19,e1 0.0,e2 0.0,e3 0.0,e4 0.0,e5 0.0,e6 0.0}
DECL FDAT FP498={TOOL_NO 1,BASE_NO 0,IPO_FRAME #BASE}
DECL PDAT PPDAT335={VEL 100.0,ACC 100.0,APO_DIST 100.0}
DECL E6POS XP499={x 2502.83008,y 203.052399,z 526.657227,a -162.090805,b 40.4880486,c -168.669601,s 6,t 19,e1 0.0,e2 0.0,e3 0.0,e4 0.0,e5 0.0,e6 0.0}
DECL FDAT FP499={TOOL_NO 1,BASE_NO 0,IPO_FRAME #BASE}
DECL LDAT LCPDAT151={VEL 2.0,ACC 100.0,APO_DIST 100.0,APO_FAC 50.0}
DECL E6POS XP500={x 2502.83496,y 203.052704,z 626.303589,a -162.090698,b 40.4886894,c -168.669403,s 6,t 19,e1 0.0,e2 0.0,e3 0.0,e4 0.0,e5 0.0,e6 0.0}
DECL FDAT FP500={TOOL_NO 1,BASE_NO 0,IPO_FRAME #BASE}
DECL LDAT LCPDAT152={VEL 2.0,ACC 100.0,APO_DIST 100.0,APO_FAC 50.0}
DECL E6POS XP501={x 2499.56299,y 91.4958115,z 626.33551,a -162.087708,b 40.4870605,c -168.667404,s 6,t 19,e1 0.0,e2 0.0,e3 0.0,e4 0.0,e5 0.0,e6 0.0}
DECL FDAT FP501={TOOL_NO 1,BASE_NO 0,IPO_FRAME #BASE}
DECL LDAT LCPDAT153={VEL 2.0,ACC 100.0,APO_DIST 100.0,APO_FAC 50.0}
DECL E6POS XP502={x 2499.55908,y 91.496048,z 526.141174,a -162.088501,b 40.4864807,c -168.668198,s 6,t 19,e1 0.0,e2 0.0,e3 0.0,e4 0.0,e5 0.0,e6 0.0}
DECL FDAT FP502={TOOL_NO 1,BASE_NO 0,IPO_FRAME #BASE}
DECL LDAT LCPDAT154={VEL 2.0,ACC 100.0,APO_DIST 100.0,APO_FAC 50.0}
DECL E6POS XP503={x 2499.55908,y 205.1315,z 526.138123,a -162.088501,b 40.4864082,c -168.668106,s 6,t 19,e1 0.0,e2 0.0,e3 0.0,e4 0.0,e5 0.0,e6 0.0}
DECL FDAT FP503={TOOL_NO 1,BASE_NO 0,IPO_FRAME #BASE}
DECL LDAT LCPDAT155={VEL 2.0,ACC 100.0,APO_DIST 100.0,APO_FAC 50.0}
DECL E6POS XP504={x 2502.88599,y 204.061905,z 625.430725,a -162.0923,b 40.4906807,c -168.671402,s 6,t 19,e1 0.0,e2 0.0,e3 0.0,e4 0.0,e5 0.0,e6 0.0}
DECL FDAT FP504={TOOL_NO 1,BASE_NO 0,IPO_FRAME #BASE}
DECL LDAT LCPDAT156={VEL 2.0,ACC 100.0,APO_DIST 100.0,APO_FAC 50.0}
DECL E6POS XP505={x 2502.88599,y 204.061905,z 625.430725,a -162.0923,b 40.4906807,c -168.671402,s 6,t 19,e1 0.0,e2 0.0,e3 0.0,e4 0.0,e5 0.0,e6 0.0}
DECL FDAT FP505={TOOL_NO 1,BASE_NO 0,IPO_FRAME #BASE}
DECL PDAT PPDAT336={VEL 100.0,ACC 100.0,APO_DIST 100.0}
DECL E6POS XP506={x 2498.04004,y 232.175797,z 673.895203,a -162.088898,b 40.4866905,c -168.667801,s 6,t 19,e1 0.0,e2 0.0,e3 0.0,e4 0.0,e5 0.0,e6 0.0}
DECL FDAT FP506={TOOL_NO 1,BASE_NO 0,IPO_FRAME #BASE}
DECL LDAT LCPDAT157={VEL 2.0,ACC 100.0,APO_DIST 100.0,APO_FAC 50.0}
DECL E6POS XP507={x 2481.65405,y -327.501709,z 670.056213,a -162.080902,b 40.4787102,c -168.671295,s 6,t 18,e1 0.0,e2 0.0,e3 0.0,e4 0.0,e5 0.0,e6 0.0}
DECL FDAT FP507={TOOL_NO 1,BASE_NO 0,IPO_FRAME #BASE}
DECL LDAT LCPDAT158={VEL 2.0,ACC 100.0,APO_DIST 100.0,APO_FAC 50.0}
DECL E6POS XP508={x 2498.75488,y 233.911697,z 672.624207,a -162.084793,b 40.4891014,c -168.665497,s 6,t 19,e1 0.0,e2 0.0,e3 0.0,e4 0.0,e5 0.0,e6 0.0}
DECL FDAT FP508={TOOL_NO 1,BASE_NO 0,IPO_FRAME #BASE}
DECL LDAT LCPDAT159={VEL 2.0,ACC 100.0,APO_DIST 100.0,APO_FAC 50.0}
DECL E6POS XP509={x 2498.75488,y 233.911697,z 672.624207,a -162.084793,b 40.4891014,c -168.665497,s 6,t 19,e1 0.0,e2 0.0,e3 0.0,e4 0.0,e5 0.0,e6 0.0}
DECL FDAT FP509={TOOL_NO 1,BASE_NO 0,IPO_FRAME #BASE}
DECL PDAT PPDAT337={VEL 100.0,ACC 100.0,APO_DIST 100.0}
DECL E6POS XP510={x 2498.73193,y 233.908798,z 1251.46399,a -162.083694,b 40.4846916,c -168.665298,s 6,t 19,e1 0.0,e2 0.0,e3 0.0,e4 0.0,e5 0.0,e6 0.0}
DECL FDAT FP510={TOOL_NO 1,BASE_NO 0,IPO_FRAME #BASE}
DECL PDAT PPDAT338={VEL 100.0,ACC 100.0,APO_DIST 100.0}
DECL E6POS XP511={x 1619.98901,y -153.192703,z 765.009583,a -90.0011063,b 60.0050812,c -89.9994965,s 6,t 18,e1 0.0,e2 0.0,e3 0.0,e4 0.0,e5 0.0,e6 0.0}
DECL FDAT FP511={TOOL_NO 1,BASE_NO 0,IPO_FRAME #BASE}
DECL PDAT PPDAT339={VEL 100.0,ACC 100.0,APO_DIST 100.0}
DECL E6POS XP512={x 1582.10706,y 59.7491913,z 765.043823,a -89.9985809,b 59.9980812,c -89.9989014,s 6,t 27,e1 0.0,e2 0.0,e3 0.0,e4 0.0,e5 0.0,e6 0.0}
DECL E6POS XP513={x 1587.93298,y 268.648193,z 763.966614,a -89.9974594,b 59.9945297,c -89.999733,s 6,t 27,e1 0.0,e2 0.0,e3 0.0,e4 0.0,e5 0.0,e6 0.0}
DECL FDAT FP513={TOOL_NO 1,BASE_NO 0,IPO_FRAME #BASE}
DECL LDAT LCPDAT160={VEL 2.0,ACC 100.0,APO_DIST 100.0,APO_FAC 50.0}
DECL E6POS XP514={x 1814.26001,y 0.00321836397,z 1214.22998,a -99.2301331,b 59.5652199,c -100.673599,s 6,t 27,e1 0.0,e2 0.0,e3 0.0,e4 0.0,e5 0.0,e6 0.0}
DECL FDAT FP514={TOOL_NO 1,BASE_NO 0,IPO_FRAME #BASE}
DECL PDAT PPDAT340={VEL 100.0,ACC 100.0,APO_DIST 100.0}
DECL E6POS XP515={x 1518.50305,y 0.00398686808,z 653.569885,a -149.876801,b -4.95594501,c 177.130295,s 2,t 11,e1 0.0,e2 0.0,e3 0.0,e4 0.0,e5 0.0,e6 0.0}
DECL FDAT FP515={TOOL_NO 1,BASE_NO 0,IPO_FRAME #BASE}
DECL PDAT PPDAT341={VEL 100.0,ACC 100.0,APO_DIST 100.0}
DECL E6POS XP516={x 1532.72498,y 0.00386148994,z 652.522827,a 27.2637005,b 2.39764094,c -178.764801,s 2,t 11,e1 0.0,e2 0.0,e3 0.0,e4 0.0,e5 0.0,e6 0.0}
DECL FDAT FP516={TOOL_NO 1,BASE_NO 0,IPO_FRAME #BASE}
DECL PDAT PPDAT342={VEL 100.0,ACC 100.0,APO_DIST 100.0}
DECL E6POS XP517={x 1554.29504,y -0.00258318405,z 489.390991,a 27.2717304,b 2.40631104,c -178.760696,s 2,t 2,e1 0.0,e2 0.0,e3 0.0,e4 0.0,e5 0.0,e6 0.0}
DECL FDAT FP517={TOOL_NO 1,BASE_NO 0,IPO_FRAME #BASE}
DECL PDAT PPDAT343={VEL 100.0,ACC 100.0,APO_DIST 100.0}
DECL E6POS XP518={x 1938.25195,y 5.26641798,z 562.713806,a -148.884293,b 35.3202286,c -161.562607,s 6,t 19,e1 0.0,e2 0.0,e3 0.0,e4 0.0,e5 0.0,e6 0.0}
DECL FDAT FP518={TOOL_NO 1,BASE_NO 0,IPO_FRAME #BASE}
DECL PDAT PPDAT344={VEL 100.0,ACC 100.0,APO_DIST 100.0}
DECL E6POS XP519={x 2003.85095,y 9.72784328,z 890.816895,a -93.417717,b 63.2684898,c -95.6996918,s 6,t 19,e1 0.0,e2 0.0,e3 0.0,e4 0.0,e5 0.0,e6 0.0}
DECL FDAT FP519={TOOL_NO 1,BASE_NO 0,IPO_FRAME #BASE}
DECL PDAT PPDAT345={VEL 100.0,ACC 100.0,APO_DIST 100.0}
DECL E6POS XP520={x 2002.78894,y 9.62718868,z 718.471313,a -99.4626694,b 62.8317909,c -102.463501,s 6,t 19,e1 0.0,e2 0.0,e3 0.0,e4 0.0,e5 0.0,e6 0.0}
DECL FDAT FP520={TOOL_NO 1,BASE_NO 0,IPO_FRAME #BASE}
DECL PDAT PPDAT346={VEL 100.0,ACC 100.0,APO_DIST 100.0}
DECL E6POS XP521={x 1980.06006,y 9.61785889,z 599.403381,a -99.4721375,b 62.8322182,c -102.473999,s 6,t 19,e1 0.0,e2 0.0,e3 0.0,e4 0.0,e5 0.0,e6 0.0}
DECL FDAT FP521={TOOL_NO 1,BASE_NO 0,IPO_FRAME #BASE}
DECL PDAT PPDAT347={VEL 100.0,ACC 100.0,APO_DIST 100.0}
DECL E6POS XP522={x 1981.26404,y 45.8989296,z 599.406982,a -99.4714279,b 62.8269806,c -102.471703,s 6,t 19,e1 0.0,e2 0.0,e3 0.0,e4 0.0,e5 0.0,e6 0.0}
DECL E6POS XP523={x 1975.06396,y 12.03901,z 599.37262,a -99.4763565,b 62.8268318,c -102.477203,s 6,t 19,e1 0.0,e2 0.0,e3 0.0,e4 0.0,e5 0.0,e6 0.0}
DECL FDAT FP523={TOOL_NO 1,BASE_NO 0,IPO_FRAME #BASE}
DECL LDAT LCPDAT161={VEL 2.0,ACC 100.0,APO_DIST 100.0,APO_FAC 50.0}
DECL E6POS XP524={x 2062.95703,y 16.9326992,z 599.429626,a -99.4677734,b 62.8305016,c -102.468697,s 6,t 19,e1 0.0,e2 0.0,e3 0.0,e4 0.0,e5 0.0,e6 0.0}
DECL E6POS XP525={x 1979.92004,y 13.0207005,z 599.417175,a -99.4695892,b 62.8309212,c -102.470703,s 6,t 19,e1 0.0,e2 0.0,e3 0.0,e4 0.0,e5 0.0,e6 0.0}
DECL FDAT FP525={TOOL_NO 1,BASE_NO 0,IPO_FRAME #BASE}
DECL LDAT LCPDAT162={VEL 2.0,ACC 100.0,APO_DIST 100.0,APO_FAC 50.0}
DECL E6POS XP526={x 604.490723,y 1038.59595,z 2477.979,a 59.7007294,b 72.3409119,c -0.0940704197,s 6,t 27,e1 0.0,e2 0.0,e3 0.0,e4 0.0,e5 0.0,e6 0.0}
DECL FDAT FP526={TOOL_NO 1,BASE_NO 0,IPO_FRAME #BASE}
DECL PDAT PPDAT348={VEL 100.0,ACC 100.0,APO_DIST 100.0}
DECL E6POS XP527={x -77.9574509,y 1211.26904,z 2377.38403,a -3.70300102,b 61.6230011,c -98.3807526,s 2,t 11,e1 0.0,e2 0.0,e3 0.0,e4 0.0,e5 0.0,e6 0.0}
DECL FDAT FP527={TOOL_NO 1,BASE_NO 0,IPO_FRAME #BASE}
DECL PDAT PPDAT349={VEL 100.0,ACC 100.0,APO_DIST 100.0}
DECL E6POS XP528={x -189.8629,y 1564.37805,z 2701.78809,a -4.38355923,b 63.0751495,c -99.1560593,s 2,t 3,e1 0.0,e2 0.0,e3 0.0,e4 0.0,e5 0.0,e6 0.0}
DECL FDAT FP528={TOOL_NO 1,BASE_NO 0,IPO_FRAME #BASE}
DECL PDAT PPDAT350={VEL 100.0,ACC 100.0,APO_DIST 100.0}
DECL E6POS XP529={x -189.873596,y 1530.55103,z 2516.77588,a -4.41487598,b 63.07827,c -99.1939926,s 2,t 3,e1 0.0,e2 0.0,e3 0.0,e4 0.0,e5 0.0,e6 0.0}
DECL FDAT FP529={TOOL_NO 1,BASE_NO 0,IPO_FRAME #BASE}
DECL PDAT PPDAT351={VEL 100.0,ACC 100.0,APO_DIST 100.0}
DECL E6POS XP530={x -189.873596,y 1530.55103,z 2516.77588,a -4.41487598,b 63.07827,c -99.1939926,s 2,t 3,e1 0.0,e2 0.0,e3 0.0,e4 0.0,e5 0.0,e6 0.0}
DECL FDAT FP530={TOOL_NO 1,BASE_NO 0,IPO_FRAME #BASE}
DECL LDAT LCPDAT163={VEL 2.0,ACC 100.0,APO_DIST 100.0,APO_FAC 50.0}
DECL E6POS XP531={x 312.673492,y 1485.46399,z 2516.78101,a -4.41415882,b 63.0783081,c -99.1930695,s 2,t 11,e1 0.0,e2 0.0,e3 0.0,e4 0.0,e5 0.0,e6 0.0}
DECL FDAT FP531={TOOL_NO 1,BASE_NO 0,IPO_FRAME #BASE}
DECL LDAT LCPDAT164={VEL 2.0,ACC 100.0,APO_DIST 100.0,APO_FAC 50.0}
DECL E6POS XP532={x 1277.37695,y -1647.69202,z 555.560974,a -99.4702835,b 62.8314781,c -102.470901,s 6,t 18,e1 0.0,e2 0.0,e3 0.0,e4 0.0,e5 0.0,e6 0.0}
DECL FDAT FP532={TOOL_NO 1,BASE_NO 0,IPO_FRAME #BASE}
DECL PDAT PPDAT352={VEL 100.0,ACC 100.0,APO_DIST 100.0}
DECL E6POS XP533={x 1559.81299,y -1647.74304,z 544.826294,a -99.4726868,b 62.830719,c -102.473099,s 6,t 50,e1 0.0,e2 0.0,e3 0.0,e4 0.0,e5 0.0,e6 0.0}
DECL E6POS XP534={x 1277.06396,y -1647.74304,z 544.823425,a -99.4731216,b 62.8311005,c -102.473503,s 6,t 18,e1 0.0,e2 0.0,e3 0.0,e4 0.0,e5 0.0,e6 0.0}
DECL FDAT FP534={TOOL_NO 1,BASE_NO 0,IPO_FRAME #BASE}
DECL LDAT LCPDAT165={VEL 2.0,ACC 100.0,APO_DIST 100.0,APO_FAC 50.0}
DECL E6POS XP535={x 1525.89197,y -1748.729,z 555.976929,a -99.4060593,b 62.8095589,c -102.402901,s 6,t 50,e1 0.0,e2 0.0,e3 0.0,e4 0.0,e5 0.0,e6 0.0}
DECL E6POS XP536={x 1276.72498,y -1647.95801,z 555.985779,a -99.4056168,b 62.8098602,c -102.402298,s 6,t 18,e1 0.0,e2 0.0,e3 0.0,e4 0.0,e5 0.0,e6 0.0}
DECL FDAT FP536={TOOL_NO 1,BASE_NO 0,IPO_FRAME #BASE}
DECL LDAT LCPDAT166={VEL 2.0,ACC 100.0,APO_DIST 100.0,APO_FAC 50.0}
DECL E6POS XP537={x 1980.16504,y 8.51173592,z 599.396179,a -126.773003,b 55.8814087,c -133.036697,s 6,t 19,e1 0.0,e2 0.0,e3 0.0,e4 0.0,e5 0.0,e6 0.0}
DECL FDAT FP537={TOOL_NO 1,BASE_NO 0,IPO_FRAME #BASE}
DECL PDAT PPDAT353={VEL 100.0,ACC 100.0,APO_DIST 100.0}
DECL E6POS XP538={x -76.1883011,y 4.23233223,z 3113.60693,a -3.17956591,b 2.1709609,c 2.83908797E-18,s 3,t 2,e1 0.0,e2 0.0,e3 0.0,e4 0.0,e5 0.0,e6 0.0}
DECL FDAT FP538={TOOL_NO 1,BASE_NO 0,IPO_FRAME #BASE}
DECL PDAT PPDAT354={VEL 100.0,ACC 100.0,APO_DIST 100.0}
DECL E6POS XP539={x -1144.34595,y 63.5694809,z 1381.62,a 176.820801,b -63.6974983,c 179.999695,s 1,t 6,e1 0.0,e2 0.0,e3 0.0,e4 0.0,e5 0.0,e6 0.0}
DECL FDAT FP539={TOOL_NO 1,BASE_NO 0,IPO_FRAME #BASE}
DECL PDAT PPDAT355={VEL 100.0,ACC 100.0,APO_DIST 100.0}
DECL E6POS XP540={x -25.2309895,y 319.093597,z 2432.13599,a -85.47995,b -70.5735321,c 0.000913246477,s 1,t 6,e1 0.0,e2 0.0,e3 0.0,e4 0.0,e5 0.0,e6 0.0}
DECL FDAT FP540={TOOL_NO 1,BASE_NO 0,IPO_FRAME #BASE}
DECL PDAT PPDAT356={VEL 100.0,ACC 100.0,APO_DIST 100.0}
DECL E6POS XP541={x -2672.1499,y -325.815796,z 1392.51196,a 6.9528451,b 86.315773,c -179.998901,s 2,t 34,e1 0.0,e2 0.0,e3 0.0,e4 0.0,e5 0.0,e6 0.0}
DECL FDAT FP541={TOOL_NO 1,BASE_NO 0,IPO_FRAME #BASE}
DECL PDAT PPDAT357={VEL 100.0,ACC 100.0,APO_DIST 100.0}
DECL E6POS XP542={x 1980.18604,y 8.32794952,z 599.398926,a -99.4719696,b 62.8320808,c -102.473999,s 6,t 19,e1 0.0,e2 0.0,e3 0.0,e4 0.0,e5 0.0,e6 0.0}
DECL FDAT FP542={TOOL_NO 1,BASE_NO 0,IPO_FRAME #BASE}
DECL PDAT PPDAT358={VEL 100.0,ACC 100.0,APO_DIST 100.0}
DECL E6POS XP543={x 2059.10693,y -21.9767303,z 560.215027,a -99.4661179,b 62.8301697,c -102.466698,s 6,t 18,e1 0.0,e2 0.0,e3 0.0,e4 0.0,e5 0.0,e6 0.0}
DECL E6POS XP544={x 2059.07593,y 43.1930618,z 560.519287,a -99.4687424,b 62.8299484,c -102.469704,s 6,t 19,e1 0.0,e2 0.0,e3 0.0,e4 0.0,e5 0.0,e6 0.0}
DECL FDAT FP544={TOOL_NO 1,BASE_NO 0,IPO_FRAME #BASE}
DECL LDAT LCPDAT167={VEL 2.0,ACC 100.0,APO_DIST 100.0,APO_FAC 50.0}
DECL E6POS XP545={x 2004.10205,y 45.1081085,z 558.627625,a -99.477623,b 62.8288689,c -102.479897,s 6,t 19,e1 0.0,e2 0.0,e3 0.0,e4 0.0,e5 0.0,e6 0.0}
DECL E6POS XP546={x 1980.84302,y 7.89386177,z 561.081177,a -99.5021973,b 62.8278008,c -102.507698,s 6,t 19,e1 0.0,e2 0.0,e3 0.0,e4 0.0,e5 0.0,e6 0.0}
DECL FDAT FP546={TOOL_NO 1,BASE_NO 0,IPO_FRAME #BASE}
DECL LDAT LCPDAT168={VEL 2.0,ACC 100.0,APO_DIST 100.0,APO_FAC 50.0}
DECL E6POS XP547={x 1980.85303,y 7.89046001,z 801.354126,a -99.5012131,b 62.8285789,c -102.506599,s 6,t 19,e1 0.0,e2 0.0,e3 0.0,e4 0.0,e5 0.0,e6 0.0}
DECL FDAT FP547={TOOL_NO 1,BASE_NO 0,IPO_FRAME #BASE}
DECL PDAT PPDAT359={VEL 100.0,ACC 100.0,APO_DIST 100.0}
DECL E6POS XP548={x 2003.84998,y -2.21163988,z 609.767395,a -93.4243011,b 63.2689514,c -95.7073364,s 6,t 18,e1 0.0,e2 0.0,e3 0.0,e4 0.0,e5 0.0,e6 0.0}
DECL FDAT FP548={TOOL_NO 1,BASE_NO 0,IPO_FRAME #BASE}
DECL PDAT PPDAT360={VEL 100.0,ACC 100.0,APO_DIST 100.0}
DECL E6POS XP549={x 1966.39795,y -49.7593307,z 612.048218,a -93.4349976,b 63.2729187,c -95.7199173,s 6,t 18,e1 0.0,e2 0.0,e3 0.0,e4 0.0,e5 0.0,e6 0.0}
DECL E6POS XP550={x 1974.14502,y -114.447403,z 618.55072,a -93.430397,b 63.2694397,c -95.7148438,s 6,t 18,e1 0.0,e2 0.0,e3 0.0,e4 0.0,e5 0.0,e6 0.0}
DECL FDAT FP550={TOOL_NO 1,BASE_NO 0,IPO_FRAME #BASE}
DECL LDAT LCPDAT169={VEL 2.0,ACC 100.0,APO_DIST 100.0,APO_FAC 50.0}
DECL E6POS XP551={x 2035.15198,y -148.424606,z 622.04248,a -93.429451,b 63.2734604,c -95.7151718,s 6,t 18,e1 0.0,e2 0.0,e3 0.0,e4 0.0,e5 0.0,e6 0.0}
DECL E6POS XP552={x 2088.70801,y -99.9511337,z 627.022705,a -93.425148,b 63.2618484,c -95.7070007,s 6,t 18,e1 0.0,e2 0.0,e3 0.0,e4 0.0,e5 0.0,e6 0.0}
DECL FDAT FP552={TOOL_NO 1,BASE_NO 0,IPO_FRAME #BASE}
DECL LDAT LCPDAT170={VEL 2.0,ACC 100.0,APO_DIST 100.0,APO_FAC 50.0}
DECL E6POS XP553={x 2074.86597,y -33.8246689,z 620.394409,a -93.4295197,b 63.2658806,c -95.7135162,s 6,t 18,e1 0.0,e2 0.0,e3 0.0,e4 0.0,e5 0.0,e6 0.0}
DECL E6POS XP554={x 2004.09302,y -2.63242292,z 607.646729,a -93.4337311,b 63.2665291,c -95.719017,s 6,t 18,e1 0.0,e2 0.0,e3 0.0,e4 0.0,e5 0.0,e6 0.0}
DECL FDAT FP554={TOOL_NO 1,BASE_NO 0,IPO_FRAME #BASE}
DECL LDAT LCPDAT171={VEL 2.0,ACC 100.0,APO_DIST 100.0,APO_FAC 50.0}
DECL E6POS XP555={x 2004.09302,y -2.63242292,z 607.646729,a -93.4337311,b 63.2665291,c -95.719017,s 6,t 18,e1 0.0,e2 0.0,e3 0.0,e4 0.0,e5 0.0,e6 0.0}
DECL FDAT FP555={TOOL_NO 1,BASE_NO 0,IPO_FRAME #BASE}
DECL PDAT PPDAT361={VEL 100.0,ACC 100.0,APO_DIST 100.0}
DECL E6POS XP556={x 2004.08496,y -2.63638711,z 964.049377,a -93.4360733,b 63.2675781,c -95.7214966,s 6,t 18,e1 0.0,e2 0.0,e3 0.0,e4 0.0,e5 0.0,e6 0.0}
DECL FDAT FP556={TOOL_NO 1,BASE_NO 0,IPO_FRAME #BASE}
DECL PDAT PPDAT362={VEL 100.0,ACC 100.0,APO_DIST 100.0}
DECL E6POS XP557={x 1814.61401,y 0.00257187197,z 1218.39099,a -99.1182785,b 63.6082382,c -100.158096,s 6,t 27,e1 0.0,e2 0.0,e3 0.0,e4 0.0,e5 0.0,e6 0.0}
DECL FDAT FP557={TOOL_NO 1,BASE_NO 0,IPO_FRAME #BASE}
DECL PDAT PPDAT363={VEL 100.0,ACC 100.0,APO_DIST 100.0}
DECL E6POS XP558={x 2056.59497,y -12.0061703,z 833.180176,a -99.118248,b 63.6088219,c -100.157501,s 6,t 18,e1 0.0,e2 0.0,e3 0.0,e4 0.0,e5 0.0,e6 0.0}
DECL FDAT FP558={TOOL_NO 1,BASE_NO 0,IPO_FRAME #BASE}
DECL PDAT PPDAT364={VEL 100.0,ACC 100.0,APO_DIST 100.0}
DECL E6POS XP559={x 2056.59912,y -12.0086203,z 771.46991,a -99.1188431,b 63.6087303,c -100.158501,s 6,t 18,e1 0.0,e2 0.0,e3 0.0,e4 0.0,e5 0.0,e6 0.0}
DECL FDAT FP559={TOOL_NO 1,BASE_NO 0,IPO_FRAME #BASE}
DECL PDAT PPDAT365={VEL 100.0,ACC 100.0,APO_DIST 100.0}
DECL E6POS XP560={x 2003.0,y -57.7944908,z 779.649414,a -99.1315079,b 63.6096802,c -100.173103,s 6,t 18,e1 0.0,e2 0.0,e3 0.0,e4 0.0,e5 0.0,e6 0.0}
DECL E6POS XP561={x 1990.06006,y -107.620003,z 778.273621,a -99.147049,b 63.6139603,c -100.192101,s 6,t 18,e1 0.0,e2 0.0,e3 0.0,e4 0.0,e5 0.0,e6 0.0}
DECL FDAT FP561={TOOL_NO 1,BASE_NO 0,IPO_FRAME #BASE}
DECL LDAT LCPDAT172={VEL 2.0,ACC 100.0,APO_DIST 100.0,APO_FAC 50.0}
DECL E6POS XP562={x 2040.08899,y -162.371994,z 783.267578,a -99.1471329,b 63.6155205,c -100.192398,s 6,t 18,e1 0.0,e2 0.0,e3 0.0,e4 0.0,e5 0.0,e6 0.0}
DECL E6POS XP563={x 2099.70996,y -132.203293,z 784.710876,a -99.1449738,b 63.6147003,c -100.189102,s 6,t 18,e1 0.0,e2 0.0,e3 0.0,e4 0.0,e5 0.0,e6 0.0}
DECL FDAT FP563={TOOL_NO 1,BASE_NO 0,IPO_FRAME #BASE}
DECL LDAT LCPDAT173={VEL 2.0,ACC 100.0,APO_DIST 100.0,APO_FAC 50.0}
DECL E6POS XP564={x 2110.66797,y -69.7507172,z 784.880798,a -99.1478119,b 63.6154213,c -100.191902,s 6,t 18,e1 0.0,e2 0.0,e3 0.0,e4 0.0,e5 0.0,e6 0.0}
DECL E6POS XP565={x 2110.66797,y -69.7507172,z 784.880798,a -99.1478119,b 63.6154213,c -100.191902,s 6,t 18,e1 0.0,e2 0.0,e3 0.0,e4 0.0,e5 0.0,e6 0.0}
DECL FDAT FP565={TOOL_NO 1,BASE_NO 0,IPO_FRAME #BASE}
DECL LDAT LCPDAT174={VEL 2.0,ACC 100.0,APO_DIST 100.0,APO_FAC 50.0}
DECL E6POS XP566={x 2094.88696,y -35.0995407,z 781.700378,a -99.140007,b 63.6152496,c -100.181503,s 6,t 18,e1 0.0,e2 0.0,e3 0.0,e4 0.0,e5 0.0,e6 0.0}
DECL E6POS XP567={x 2057.10205,y -12.5491896,z 771.215698,a -99.1455307,b 63.6152496,c -100.187103,s 6,t 18,e1 0.0,e2 0.0,e3 0.0,e4 0.0,e5 0.0,e6 0.0}
DECL FDAT FP567={TOOL_NO 1,BASE_NO 0,IPO_FRAME #BASE}
DECL LDAT LCPDAT175={VEL 2.0,ACC 100.0,APO_DIST 100.0,APO_FAC 50.0}
DECL E6POS XP568={x 2057.10205,y -12.5491896,z 771.215698,a -99.1455307,b 63.6152496,c -100.187103,s 6,t 18,e1 0.0,e2 0.0,e3 0.0,e4 0.0,e5 0.0,e6 0.0}
DECL FDAT FP568={TOOL_NO 1,BASE_NO 0,IPO_FRAME #BASE}
DECL PDAT PPDAT366={VEL 100.0,ACC 100.0,APO_DIST 100.0}
DECL E6POS XP569={x 2057.10889,y -12.5443897,z 1051.78003,a -99.1448669,b 63.6157303,c -100.1866,s 6,t 18,e1 0.0,e2 0.0,e3 0.0,e4 0.0,e5 0.0,e6 0.0}
DECL FDAT FP569={TOOL_NO 1,BASE_NO 0,IPO_FRAME #BASE}
DECL PDAT PPDAT367={VEL 100.0,ACC 100.0,APO_DIST 100.0}
DECL E6POS XP570={x 691.286621,y -34.6563797,z 1515.48999,a -157.6026,b -4.36903,c 178.825806,s 2,t 2,e1 0.0,e2 0.0,e3 0.0,e4 0.0,e5 0.0,e6 0.0}
DECL FDAT FP570={TOOL_NO 1,BASE_NO 0,IPO_FRAME #BASE}
DECL PDAT PPDAT368={VEL 100.0,ACC 100.0,APO_DIST 100.0}
DECL E6POS XP571={x 691.434509,y -30.9982891,z 1515.453,a -157.762497,b -4.04829216,c 178.131805,s 2,t 2,e1 0.0,e2 0.0,e3 0.0,e4 0.0,e5 0.0,e6 0.0}
DECL FDAT FP571={TOOL_NO 1,BASE_NO 0,IPO_FRAME #BASE}
DECL PDAT PPDAT369={VEL 100.0,ACC 100.0,APO_DIST 100.0}
DECL E6POS XP572={x 1259.39294,y -56.4598389,z 1821.02905,a -157.767502,b 3.90171003,c -178.198502,s 2,t 2,e1 0.0,e2 0.0,e3 0.0,e4 0.0,e5 0.0,e6 0.0}
DECL FDAT FP572={TOOL_NO 1,BASE_NO 0,IPO_FRAME #BASE}
DECL PDAT PPDAT370={VEL 100.0,ACC 100.0,APO_DIST 100.0}
DECL E6POS XP573={x 1259.39294,y -56.4598389,z 1821.02905,a -157.767502,b 3.90171003,c -178.198502,s 2,t 2,e1 0.0,e2 0.0,e3 0.0,e4 0.0,e5 0.0,e6 0.0}
DECL FDAT FP573={TOOL_NO 1,BASE_NO 0,IPO_FRAME #BASE}
DECL PDAT PPDAT371={VEL 100.0,ACC 100.0,APO_DIST 100.0}
DECL E6POS XP574={x 1650.33203,y -0.0238221399,z 1155.71594,a -100.055,b 63.2422218,c -101.231598,s 6,t 18,e1 0.0,e2 0.0,e3 0.0,e4 0.0,e5 0.0,e6 0.0}
DECL FDAT FP574={TOOL_NO 1,BASE_NO 0,IPO_FRAME #BASE}
DECL PDAT PPDAT372={VEL 100.0,ACC 100.0,APO_DIST 100.0}
DECL E6POS XP575={x 1697.49695,y -0.0835798979,z 815.637512,a -100.057404,b 63.2419205,c -101.234703,s 6,t 18,e1 0.0,e2 0.0,e3 0.0,e4 0.0,e5 0.0,e6 0.0}
DECL FDAT FP575={TOOL_NO 1,BASE_NO 0,IPO_FRAME #BASE}
DECL PDAT PPDAT373={VEL 100.0,ACC 100.0,APO_DIST 100.0}
DECL E6POS XP576={x 1686.23999,y -0.0845535025,z 925.313721,a -100.064499,b 63.2399788,c -101.242401,s 6,t 18,e1 0.0,e2 0.0,e3 0.0,e4 0.0,e5 0.0,e6 0.0}
DECL FDAT FP576={TOOL_NO 1,BASE_NO 0,IPO_FRAME #BASE}
DECL PDAT PPDAT374={VEL 100.0,ACC 100.0,APO_DIST 100.0}
DECL E6POS XP577={x 1619.93103,y 9.73077106,z 791.904114,a -100.064201,b 63.2395096,c -101.241798,s 6,t 27,e1 0.0,e2 0.0,e3 0.0,e4 0.0,e5 0.0,e6 0.0}
DECL FDAT FP577={TOOL_NO 1,BASE_NO 0,IPO_FRAME #BASE}
DECL PDAT PPDAT375={VEL 100.0,ACC 100.0,APO_DIST 100.0}
DECL E6POS XP578={x 1645.80701,y -50.2456284,z 791.89502,a -100.066399,b 63.2396812,c -101.244202,s 6,t 18,e1 0.0,e2 0.0,e3 0.0,e4 0.0,e5 0.0,e6 0.0}
DECL E6POS XP579={x 1710.79004,y -67.8860474,z 791.892212,a -100.067398,b 63.2389107,c -101.245598,s 6,t 18,e1 0.0,e2 0.0,e3 0.0,e4 0.0,e5 0.0,e6 0.0}
DECL FDAT FP579={TOOL_NO 1,BASE_NO 0,IPO_FRAME #BASE}
DECL LDAT LCPDAT176={VEL 2.0,ACC 100.0,APO_DIST 100.0,APO_FAC 50.0}
DECL E6POS XP580={x 1735.59998,y -46.3213806,z 791.902771,a -100.066803,b 63.2386703,c -101.244904,s 6,t 18,e1 0.0,e2 0.0,e3 0.0,e4 0.0,e5 0.0,e6 0.0}
DECL E6POS XP581={x 1752.02295,y 18.9178905,z 791.906006,a -100.066902,b 63.2383919,c -101.244598,s 6,t 27,e1 0.0,e2 0.0,e3 0.0,e4 0.0,e5 0.0,e6 0.0}
DECL FDAT FP581={TOOL_NO 1,BASE_NO 0,IPO_FRAME #BASE}
DECL LDAT LCPDAT177={VEL 2.0,ACC 100.0,APO_DIST 100.0,APO_FAC 50.0}
DECL E6POS XP583={x 1697.10999,y 62.8259315,z 791.899475,a -100.068398,b 63.2375908,c -101.245903,s 6,t 27,e1 0.0,e2 0.0,e3 0.0,e4 0.0,e5 0.0,e6 0.0}
DECL E6POS XP582={x 1698.77002,y 19.32971,z 771.787292,a -100.069504,b 63.2397995,c -101.248299,s 6,t 27,e1 0.0,e2 0.0,e3 0.0,e4 0.0,e5 0.0,e6 0.0}
DECL FDAT FP582={TOOL_NO 1,BASE_NO 0,IPO_FRAME #BASE}
DECL PDAT PPDAT376={VEL 100.0,ACC 100.0,APO_DIST 100.0}
DECL E6POS XP584={x 1698.78003,y 19.3298397,z 771.789978,a -100.068398,b 63.2399101,c -101.247002,s 6,t 27,e1 0.0,e2 0.0,e3 0.0,e4 0.0,e5 0.0,e6 0.0}
DECL FDAT FP584={TOOL_NO 1,BASE_NO 0,IPO_FRAME #BASE}
DECL PDAT PPDAT377={VEL 100.0,ACC 100.0,APO_DIST 100.0}
DECL E6POS XP585={x 2337.92505,y -0.0893416405,z 570.093384,a -153.627594,b -3.78119898,c 178.129501,s 2,t 2,e1 0.0,e2 0.0,e3 0.0,e4 0.0,e5 0.0,e6 0.0}
DECL FDAT FP585={TOOL_NO 1,BASE_NO 0,IPO_FRAME #BASE}
DECL PDAT PPDAT378={VEL 100.0,ACC 100.0,APO_DIST 100.0}
DECL E6POS XP586={x 2337.88892,y -0.0889165103,z 243.5354,a -153.626999,b -3.78581905,c 178.126999,s 2,t 0,e1 0.0,e2 0.0,e3 0.0,e4 0.0,e5 0.0,e6 0.0}
DECL FDAT FP586={TOOL_NO 1,BASE_NO 0,IPO_FRAME #BASE}
DECL PDAT PPDAT379={VEL 100.0,ACC 100.0,APO_DIST 100.0}
DECL E6POS XP587={x 2253.64111,y -0.0903828815,z 264.990112,a -153.615799,b -3.82170391,c 178.108307,s 2,t 2,e1 0.0,e2 0.0,e3 0.0,e4 0.0,e5 0.0,e6 0.0}
DECL FDAT FP587={TOOL_NO 1,BASE_NO 0,IPO_FRAME #BASE}
DECL PDAT PPDAT380={VEL 100.0,ACC 100.0,APO_DIST 100.0}
DECL E6POS XP588={x 2253.64111,y -0.0903828815,z 264.990112,a -153.615799,b -3.82170391,c 178.108307,s 2,t 2,e1 0.0,e2 0.0,e3 0.0,e4 0.0,e5 0.0,e6 0.0}
DECL FDAT FP588={TOOL_NO 1,BASE_NO 0,IPO_FRAME #BASE}
DECL LDAT LCPDAT178={VEL 2.0,ACC 100.0,APO_DIST 100.0,APO_FAC 50.0}
DECL E6POS XP589={x 2253.85498,y -17.1867809,z 214.235199,a -153.612396,b -3.83106208,c 178.103394,s 2,t 2,e1 0.0,e2 0.0,e3 0.0,e4 0.0,e5 0.0,e6 0.0}
DECL FDAT FP589={TOOL_NO 1,BASE_NO 0,IPO_FRAME #BASE}
DECL LDAT LCPDAT179={VEL 2.0,ACC 100.0,APO_DIST 100.0,APO_FAC 50.0}
DECL E6POS XP590={x 2261.06104,y 16.4479504,z 213.942795,a -153.612396,b -3.84011102,c 178.099304,s 2,t 11,e1 0.0,e2 0.0,e3 0.0,e4 0.0,e5 0.0,e6 0.0}
DECL FDAT FP590={TOOL_NO 1,BASE_NO 0,IPO_FRAME #BASE}
DECL LDAT LCPDAT180={VEL 2.0,ACC 100.0,APO_DIST 100.0,APO_FAC 50.0}
DECL E6POS XP591={x 2252.31592,y -0.362133414,z 263.964813,a -153.6082,b -3.85193205,c 178.093002,s 2,t 2,e1 0.0,e2 0.0,e3 0.0,e4 0.0,e5 0.0,e6 0.0}
DECL FDAT FP591={TOOL_NO 1,BASE_NO 0,IPO_FRAME #BASE}
DECL LDAT LCPDAT181={VEL 2.0,ACC 100.0,APO_DIST 100.0,APO_FAC 50.0}
DECL E6POS XP592={x 2252.31592,y -0.362133414,z 263.964813,a -153.6082,b -3.85193205,c 178.093002,s 2,t 2,e1 0.0,e2 0.0,e3 0.0,e4 0.0,e5 0.0,e6 0.0}
DECL FDAT FP592={TOOL_NO 1,BASE_NO 0,IPO_FRAME #BASE}
DECL PDAT PPDAT381={VEL 100.0,ACC 100.0,APO_DIST 100.0}
DECL E6POS XP593={x 2386.79199,y -0.361944109,z 263.21051,a -153.610504,b -3.84308004,c 178.097504,s 2,t 0,e1 0.0,e2 0.0,e3 0.0,e4 0.0,e5 0.0,e6 0.0}
DECL FDAT FP593={TOOL_NO 1,BASE_NO 0,IPO_FRAME #BASE}
DECL PDAT PPDAT382={VEL 100.0,ACC 100.0,APO_DIST 100.0}
DECL E6POS XP594={x 2493.60498,y -0.0846298933,z 1014.91602,a -100.070198,b 63.2411385,c -101.248802,s 6,t 18,e1 0.0,e2 0.0,e3 0.0,e4 0.0,e5 0.0,e6 0.0}
DECL FDAT FP594={TOOL_NO 1,BASE_NO 0,IPO_FRAME #BASE}
DECL PDAT PPDAT383={VEL 100.0,ACC 100.0,APO_DIST 100.0}
DECL E6POS XP595={x 2410.39502,y -18.5170708,z 282.790405,a -153.605301,b -3.83601093,c 178.099792,s 2,t 0,e1 0.0,e2 0.0,e3 0.0,e4 0.0,e5 0.0,e6 0.0}
DECL FDAT FP595={TOOL_NO 1,BASE_NO 0,IPO_FRAME #BASE}
DECL PDAT PPDAT384={VEL 100.0,ACC 100.0,APO_DIST 100.0}
DECL E6POS XP596={x 2272.37793,y -18.4971409,z 282.600311,a -153.603195,b -3.83755112,c 178.098602,s 2,t 2,e1 0.0,e2 0.0,e3 0.0,e4 0.0,e5 0.0,e6 0.0}
DECL FDAT FP596={TOOL_NO 1,BASE_NO 0,IPO_FRAME #BASE}
DECL PDAT PPDAT385={VEL 100.0,ACC 100.0,APO_DIST 100.0}
DECL E6POS XP597={x 2272.37793,y -18.4971409,z 282.600311,a -153.603195,b -3.83755112,c 178.098602,s 2,t 2,e1 0.0,e2 0.0,e3 0.0,e4 0.0,e5 0.0,e6 0.0}
DECL FDAT FP597={TOOL_NO 1,BASE_NO 0,IPO_FRAME #BASE}
DECL PDAT PPDAT386={VEL 100.0,ACC 100.0,APO_DIST 100.0}
DECL E6POS XP598={x 2238.68506,y -18.4194298,z 281.963196,a -153.5961,b -3.85345602,c 178.089294,s 2,t 2,e1 0.0,e2 0.0,e3 0.0,e4 0.0,e5 0.0,e6 0.0}
DECL FDAT FP598={TOOL_NO 1,BASE_NO 0,IPO_FRAME #BASE}
DECL PDAT PPDAT387={VEL 100.0,ACC 100.0,APO_DIST 100.0}
DECL E6POS XP599={x 2238.68506,y -18.4194298,z 281.963196,a -153.5961,b -3.85345602,c 178.089294,s 2,t 2,e1 0.0,e2 0.0,e3 0.0,e4 0.0,e5 0.0,e6 0.0}
DECL FDAT FP599={TOOL_NO 1,BASE_NO 0,IPO_FRAME #BASE}
DECL LDAT LCPDAT182={VEL 2.0,ACC 100.0,APO_DIST 100.0,APO_FAC 50.0}
DECL E6POS XP600={x 2223.54712,y -69.8122864,z 261.026611,a -153.591599,b -3.86129594,c 178.083801,s 2,t 2,e1 0.0,e2 0.0,e3 0.0,e4 0.0,e5 0.0,e6 0.0}
DECL FDAT FP600={TOOL_NO 1,BASE_NO 0,IPO_FRAME #BASE}
DECL LDAT LCPDAT183={VEL 2.0,ACC 100.0,APO_DIST 100.0,APO_FAC 50.0}
DECL E6POS XP601={x 2237.62598,y -49.5636292,z 242.4198,a -153.588806,b -3.86524105,c 178.081604,s 2,t 2,e1 0.0,e2 0.0,e3 0.0,e4 0.0,e5 0.0,e6 0.0}
DECL FDAT FP601={TOOL_NO 1,BASE_NO 0,IPO_FRAME #BASE}
DECL LDAT LCPDAT184={VEL 2.0,ACC 100.0,APO_DIST 100.0,APO_FAC 50.0}
DECL E6POS XP602={x 2237.71094,y -18.7772808,z 281.085388,a -153.585403,b -3.87217402,c 178.078201,s 2,t 2,e1 0.0,e2 0.0,e3 0.0,e4 0.0,e5 0.0,e6 0.0}
DECL FDAT FP602={TOOL_NO 1,BASE_NO 0,IPO_FRAME #BASE}
DECL LDAT LCPDAT185={VEL 2.0,ACC 100.0,APO_DIST 100.0,APO_FAC 50.0}
DECL E6POS XP603={x 2237.71094,y -18.7772808,z 281.085388,a -153.585403,b -3.87217402,c 178.078201,s 2,t 2,e1 0.0,e2 0.0,e3 0.0,e4 0.0,e5 0.0,e6 0.0}
DECL FDAT FP603={TOOL_NO 1,BASE_NO 0,IPO_FRAME #BASE}
DECL PDAT PPDAT388={VEL 100.0,ACC 100.0,APO_DIST 100.0}
DECL E6POS XP604={x 2358.64893,y -18.7991104,z 281.101501,a -153.588303,b -3.86433101,c 178.082703,s 2,t 2,e1 0.0,e2 0.0,e3 0.0,e4 0.0,e5 0.0,e6 0.0}
DECL FDAT FP604={TOOL_NO 1,BASE_NO 0,IPO_FRAME #BASE}
DECL PDAT PPDAT389={VEL 100.0,ACC 100.0,APO_DIST 100.0}
DECL E6POS XP605={x 2370.95093,y 17.5828705,z 282.17981,a -153.587402,b -3.87034106,c 178.079697,s 2,t 9,e1 0.0,e2 0.0,e3 0.0,e4 0.0,e5 0.0,e6 0.0}
DECL FDAT FP605={TOOL_NO 1,BASE_NO 0,IPO_FRAME #BASE}
DECL PDAT PPDAT390={VEL 100.0,ACC 100.0,APO_DIST 100.0}
DECL E6POS XP606={x 2268.63696,y 17.5842991,z 282.156311,a -153.587006,b -3.87018609,c 178.079697,s 2,t 11,e1 0.0,e2 0.0,e3 0.0,e4 0.0,e5 0.0,e6 0.0}
DECL FDAT FP606={TOOL_NO 1,BASE_NO 0,IPO_FRAME #BASE}
DECL PDAT PPDAT391={VEL 100.0,ACC 100.0,APO_DIST 100.0}
DECL E6POS XP607={x 2237.552,y 17.5505199,z 281.76239,a -153.583893,b -3.8816359,c 178.074203,s 2,t 11,e1 0.0,e2 0.0,e3 0.0,e4 0.0,e5 0.0,e6 0.0}
DECL FDAT FP607={TOOL_NO 1,BASE_NO 0,IPO_FRAME #BASE}
DECL PDAT PPDAT392={VEL 100.0,ACC 100.0,APO_DIST 100.0}
DECL E6POS XP608={x 2237.552,y 17.5505199,z 281.76239,a -153.583893,b -3.8816359,c 178.074203,s 2,t 11,e1 0.0,e2 0.0,e3 0.0,e4 0.0,e5 0.0,e6 0.0}
DECL FDAT FP608={TOOL_NO 1,BASE_NO 0,IPO_FRAME #BASE}
DECL LDAT LCPDAT186={VEL 2.0,ACC 100.0,APO_DIST 100.0,APO_FAC 50.0}
DECL E6POS XP609={x 2249.32202,y 64.8089523,z 241.657593,a -153.585297,b -3.8850379,c 178.073395,s 2,t 11,e1 0.0,e2 0.0,e3 0.0,e4 0.0,e5 0.0,e6 0.0}
DECL FDAT FP609={TOOL_NO 1,BASE_NO 0,IPO_FRAME #BASE}
DECL LDAT LCPDAT187={VEL 2.0,ACC 100.0,APO_DIST 100.0,APO_FAC 50.0}
DECL E6POS XP610={x 2231.93799,y 73.8221512,z 271.105713,a -153.581894,b -3.89104009,c 178.071304,s 2,t 11,e1 0.0,e2 0.0,e3 0.0,e4 0.0,e5 0.0,e6 0.0}
DECL FDAT FP610={TOOL_NO 1,BASE_NO 0,IPO_FRAME #BASE}
DECL LDAT LCPDAT188={VEL 2.0,ACC 100.0,APO_DIST 100.0,APO_FAC 50.0}
DECL E6POS XP611={x 2238.23804,y 17.1711006,z 281.552399,a -153.576996,b -3.90073204,c 178.065704,s 2,t 11,e1 0.0,e2 0.0,e3 0.0,e4 0.0,e5 0.0,e6 0.0}
DECL FDAT FP611={TOOL_NO 1,BASE_NO 0,IPO_FRAME #BASE}
DECL LDAT LCPDAT189={VEL 2.0,ACC 100.0,APO_DIST 100.0,APO_FAC 50.0}
DECL E6POS XP612={x 2238.23804,y 17.1711006,z 281.552399,a -153.576996,b -3.90073204,c 178.065704,s 2,t 11,e1 0.0,e2 0.0,e3 0.0,e4 0.0,e5 0.0,e6 0.0}
DECL FDAT FP612={TOOL_NO 1,BASE_NO 0,IPO_FRAME #BASE}
DECL PDAT PPDAT393={VEL 100.0,ACC 100.0,APO_DIST 100.0}
DECL E6POS XP613={x 2270.05688,y 17.1765194,z 281.452209,a -153.578003,b -3.90055895,c 178.065399,s 2,t 11,e1 0.0,e2 0.0,e3 0.0,e4 0.0,e5 0.0,e6 0.0}
DECL FDAT FP613={TOOL_NO 1,BASE_NO 0,IPO_FRAME #BASE}
DECL PDAT PPDAT394={VEL 100.0,ACC 100.0,APO_DIST 100.0}
DECL E6POS XP614={x 2384.36792,y 17.1860809,z 281.477905,a -153.5793,b -3.89311194,c 178.069199,s 2,t 9,e1 0.0,e2 0.0,e3 0.0,e4 0.0,e5 0.0,e6 0.0}
DECL FDAT FP614={TOOL_NO 1,BASE_NO 0,IPO_FRAME #BASE}
DECL PDAT PPDAT395={VEL 100.0,ACC 100.0,APO_DIST 100.0}
DECL E6POS XP615={x 2375.61597,y -75.9825974,z 200.707306,a -153.580093,b -3.88543391,c 178.072906,s 2,t 0,e1 0.0,e2 0.0,e3 0.0,e4 0.0,e5 0.0,e6 0.0}
DECL FDAT FP615={TOOL_NO 1,BASE_NO 0,IPO_FRAME #BASE}
DECL PDAT PPDAT396={VEL 100.0,ACC 100.0,APO_DIST 100.0}
DECL E6POS XP616={x 2260.13501,y -75.7760162,z 200.315506,a -153.571396,b -3.9083271,c 178.058304,s 2,t 2,e1 0.0,e2 0.0,e3 0.0,e4 0.0,e5 0.0,e6 0.0}
DECL FDAT FP616={TOOL_NO 1,BASE_NO 0,IPO_FRAME #BASE}
DECL PDAT PPDAT397={VEL 100.0,ACC 100.0,APO_DIST 100.0}
DECL E6POS XP617={x 2233.55688,y -75.5832367,z 199.812103,a -153.565506,b -3.91943097,c 178.050705,s 2,t 2,e1 0.0,e2 0.0,e3 0.0,e4 0.0,e5 0.0,e6 0.0}
DECL FDAT FP617={TOOL_NO 1,BASE_NO 0,IPO_FRAME #BASE}
DECL PDAT PPDAT398={VEL 100.0,ACC 100.0,APO_DIST 100.0}
DECL E6POS XP618={x 2233.55688,y -75.5832367,z 199.812103,a -153.565506,b -3.91943097,c 178.050705,s 2,t 2,e1 0.0,e2 0.0,e3 0.0,e4 0.0,e5 0.0,e6 0.0}
DECL FDAT FP618={TOOL_NO 1,BASE_NO 0,IPO_FRAME #BASE}
DECL LDAT LCPDAT190={VEL 2.0,ACC 100.0,APO_DIST 100.0,APO_FAC 50.0}
DECL E6POS XP619={x 2248.03906,y -31.169241,z 167.907593,a -153.565002,b -3.9285419,c 178.046494,s 2,t 2,e1 0.0,e2 0.0,e3 0.0,e4 0.0,e5 0.0,e6 0.0}
DECL FDAT FP619={TOOL_NO 1,BASE_NO 0,IPO_FRAME #BASE}
DECL LDAT LCPDAT191={VEL 2.0,ACC 100.0,APO_DIST 100.0,APO_FAC 50.0}
DECL E6POS XP620={x 2258.29297,y 9.88335419,z 167.974304,a -153.567703,b -3.93106103,c 178.045807,s 2,t 11,e1 0.0,e2 0.0,e3 0.0,e4 0.0,e5 0.0,e6 0.0}
DECL FDAT FP620={TOOL_NO 1,BASE_NO 0,IPO_FRAME #BASE}
DECL LDAT LCPDAT192={VEL 2.0,ACC 100.0,APO_DIST 100.0,APO_FAC 50.0}
DECL E6POS XP621={x 2260.74292,y 9.87940884,z 180.593796,a -153.566895,b -3.92987895,c 178.046295,s 2,t 11,e1 0.0,e2 0.0,e3 0.0,e4 0.0,e5 0.0,e6 0.0}
DECL FDAT FP621={TOOL_NO 1,BASE_NO 0,IPO_FRAME #BASE}
DECL LDAT LCPDAT193={VEL 2.0,ACC 100.0,APO_DIST 100.0,APO_FAC 50.0}
DECL E6POS XP622={x 2259.93896,y 29.6603508,z 183.124207,a -153.565796,b -3.93438196,c 178.044693,s 2,t 11,e1 0.0,e2 0.0,e3 0.0,e4 0.0,e5 0.0,e6 0.0}
DECL FDAT FP622={TOOL_NO 1,BASE_NO 0,IPO_FRAME #BASE}
DECL LDAT LCPDAT194={VEL 2.0,ACC 100.0,APO_DIST 100.0,APO_FAC 50.0}
DECL E6POS XP623={x 2254.1499,y 31.82938,z 173.739502,a -153.560394,b -3.94960093,c 178.037598,s 2,t 11,e1 0.0,e2 0.0,e3 0.0,e4 0.0,e5 0.0,e6 0.0}
DECL FDAT FP623={TOOL_NO 1,BASE_NO 0,IPO_FRAME #BASE}
DECL LDAT LCPDAT195={VEL 2.0,ACC 100.0,APO_DIST 100.0,APO_FAC 50.0}
DECL E6POS XP624={x 2252.229,y 42.4542618,z 173.891205,a -153.561707,b -3.94484901,c 178.039993,s 2,t 11,e1 0.0,e2 0.0,e3 0.0,e4 0.0,e5 0.0,e6 0.0}
DECL FDAT FP624={TOOL_NO 1,BASE_NO 0,IPO_FRAME #BASE}
DECL LDAT LCPDAT196={VEL 2.0,ACC 100.0,APO_DIST 100.0,APO_FAC 50.0}
DECL E6POS XP625={x 2246.98608,y 85.3690414,z 208.387497,a -153.560806,b -3.94197989,c 178.042603,s 2,t 11,e1 0.0,e2 0.0,e3 0.0,e4 0.0,e5 0.0,e6 0.0}
DECL FDAT FP625={TOOL_NO 1,BASE_NO 0,IPO_FRAME #BASE}
DECL LDAT LCPDAT197={VEL 2.0,ACC 100.0,APO_DIST 100.0,APO_FAC 50.0}
DECL E6POS XP626={x 2261.14502,y 35.6814804,z 195.084,a -153.561295,b -3.94195795,c 178.041901,s 2,t 11,e1 0.0,e2 0.0,e3 0.0,e4 0.0,e5 0.0,e6 0.0}
DECL FDAT FP626={TOOL_NO 1,BASE_NO 0,IPO_FRAME #BASE}
DECL LDAT LCPDAT198={VEL 2.0,ACC 100.0,APO_DIST 100.0,APO_FAC 50.0}
DECL E6POS XP627={x 2259.39404,y -1.94677496,z 191.305695,a -153.558899,b -3.94204307,c 178.040802,s 2,t 2,e1 0.0,e2 0.0,e3 0.0,e4 0.0,e5 0.0,e6 0.0}
DECL FDAT FP627={TOOL_NO 1,BASE_NO 0,IPO_FRAME #BASE}
DECL LDAT LCPDAT199={VEL 2.0,ACC 100.0,APO_DIST 100.0,APO_FAC 50.0}
DECL E6POS XP628={x 2254.30908,y -1.95780003,z 180.317093,a -153.559998,b -3.93576002,c 178.044205,s 2,t 2,e1 0.0,e2 0.0,e3 0.0,e4 0.0,e5 0.0,e6 0.0}
DECL FDAT FP628={TOOL_NO 1,BASE_NO 0,IPO_FRAME #BASE}
DECL LDAT LCPDAT200={VEL 2.0,ACC 100.0,APO_DIST 100.0,APO_FAC 50.0}
DECL E6POS XP629={x 2251.70288,y -26.0037403,z 180.578506,a -153.563095,b -3.93059611,c 178.046906,s 2,t 2,e1 0.0,e2 0.0,e3 0.0,e4 0.0,e5 0.0,e6 0.0}
DECL FDAT FP629={TOOL_NO 1,BASE_NO 0,IPO_FRAME #BASE}
DECL LDAT LCPDAT201={VEL 2.0,ACC 100.0,APO_DIST 100.0,APO_FAC 50.0}
DECL E6POS XP630={x 2259.4231,y -26.9836197,z 191.557602,a -153.564194,b -3.9261241,c 178.049393,s 2,t 2,e1 0.0,e2 0.0,e3 0.0,e4 0.0,e5 0.0,e6 0.0}
DECL FDAT FP630={TOOL_NO 1,BASE_NO 0,IPO_FRAME #BASE}
DECL LDAT LCPDAT202={VEL 2.0,ACC 100.0,APO_DIST 100.0,APO_FAC 50.0}
DECL E6POS XP631={x 2232.13989,y -76.6630478,z 200.910294,a -153.564896,b -3.92678189,c 178.048294,s 2,t 2,e1 0.0,e2 0.0,e3 0.0,e4 0.0,e5 0.0,e6 0.0}
DECL FDAT FP631={TOOL_NO 1,BASE_NO 0,IPO_FRAME #BASE}
DECL LDAT LCPDAT203={VEL 2.0,ACC 100.0,APO_DIST 100.0,APO_FAC 50.0}
DECL E6POS XP632={x 2255.46997,y -76.7131271,z 201.019104,a -153.5672,b -3.920259,c 178.052307,s 2,t 2,e1 0.0,e2 0.0,e3 0.0,e4 0.0,e5 0.0,e6 0.0}
DECL FDAT FP632={TOOL_NO 1,BASE_NO 0,IPO_FRAME #BASE}
DECL PDAT PPDAT399={VEL 100.0,ACC 100.0,APO_DIST 100.0}
DECL E6POS XP633={x 2310.23193,y -76.7230301,z 201.095093,a -153.5681,b -3.92067194,c 178.051605,s 2,t 0,e1 0.0,e2 0.0,e3 0.0,e4 0.0,e5 0.0,e6 0.0}
DECL FDAT FP633={TOOL_NO 1,BASE_NO 0,IPO_FRAME #BASE}
DECL PDAT PPDAT400={VEL 100.0,ACC 100.0,APO_DIST 100.0}
DECL E6POS XP634={x 2183.37402,y 38.41996,z 249.258499,a -153.023407,b 4.71550894,c -177.9599,s 2,t 11,e1 0.0,e2 0.0,e3 0.0,e4 0.0,e5 0.0,e6 0.0}
DECL FDAT FP634={TOOL_NO 1,BASE_NO 0,IPO_FRAME #BASE}
DECL PDAT PPDAT401={VEL 100.0,ACC 100.0,APO_DIST 100.0}
DECL E6POS XP635={x 2674.19507,y 61.8912811,z 1058.31604,a -147.084793,b 47.5691719,c -158.968399,s 2,t 11,e1 0.0,e2 0.0,e3 0.0,e4 0.0,e5 0.0,e6 0.0}
DECL FDAT FP635={TOOL_NO 1,BASE_NO 0,IPO_FRAME #BASE}
DECL PDAT PPDAT402={VEL 100.0,ACC 100.0,APO_DIST 100.0}
DECL E6POS XP636={x 2255.16602,y -1438.53796,z 1058.32605,a 179.056,b 47.5698891,c -158.968307,s 2,t 10,e1 0.0,e2 0.0,e3 0.0,e4 0.0,e5 0.0,e6 0.0}
DECL FDAT FP636={TOOL_NO 1,BASE_NO 0,IPO_FRAME #BASE}
DECL PDAT PPDAT403={VEL 100.0,ACC 100.0,APO_DIST 100.0}
DECL E6POS XP637={x 1963.09802,y -1242.99304,z 504.068298,a 169.090195,b 5.26360893,c 177.121994,s 2,t 10,e1 0.0,e2 0.0,e3 0.0,e4 0.0,e5 0.0,e6 0.0}
DECL FDAT FP637={TOOL_NO 1,BASE_NO 0,IPO_FRAME #BASE}
DECL PDAT PPDAT404={VEL 100.0,ACC 100.0,APO_DIST 100.0}
DECL E6POS XP638={x 1963.09998,y -1242.99304,z 1467.72803,a 169.090302,b 5.26396704,c 177.122101,s 2,t 10,e1 0.0,e2 0.0,e3 0.0,e4 0.0,e5 0.0,e6 0.0}
DECL FDAT FP638={TOOL_NO 1,BASE_NO 0,IPO_FRAME #BASE}
DECL PDAT PPDAT405={VEL 100.0,ACC 100.0,APO_DIST 100.0}
DECL E6POS XP639={x -1376.89197,y -1798.63403,z 1948.46399,a 133.761398,b 72.5001831,c -99.2481003,s 2,t 10,e1 0.0,e2 0.0,e3 0.0,e4 0.0,e5 0.0,e6 0.0}
DECL FDAT FP639={TOOL_NO 1,BASE_NO 0,IPO_FRAME #BASE}
DECL PDAT PPDAT406={VEL 100.0,ACC 100.0,APO_DIST 100.0}
DECL E6POS XP640={x 1863.23706,y -870.91449,z 2259.24609,a -91.1544266,b 71.0322418,c -64.9191589,s 2,t 10,e1 0.0,e2 0.0,e3 0.0,e4 0.0,e5 0.0,e6 0.0}
DECL FDAT FP640={TOOL_NO 1,BASE_NO 0,IPO_FRAME #BASE}
DECL PDAT PPDAT407={VEL 100.0,ACC 100.0,APO_DIST 100.0}
DECL E6POS XP641={x 428.551514,y -0.0108004203,z 3259.09692,a -17.3059196,b -0.494722605,c 0.126435801,s 0,t 14,e1 0.0,e2 0.0,e3 0.0,e4 0.0,e5 0.0,e6 0.0}
DECL FDAT FP641={TOOL_NO 1,BASE_NO 0,IPO_FRAME #BASE}
DECL PDAT PPDAT408={VEL 100.0,ACC 100.0,APO_DIST 100.0}
DECL E6POS XP642={x -1330.20996,y 0.541942775,z 1791.36304,a -96.7218933,b -72.5895309,c 96.9951019,s 1,t 14,e1 0.0,e2 0.0,e3 0.0,e4 0.0,e5 0.0,e6 0.0}
DECL FDAT FP642={TOOL_NO 1,BASE_NO 0,IPO_FRAME #BASE}
DECL PDAT PPDAT409={VEL 100.0,ACC 100.0,APO_DIST 100.0}
DECL E6POS XP643={x 115.931702,y -368.9086,z 3258.39111,a -89.8604889,b -0.196505293,c 0.0336363986,s 0,t 10,e1 0.0,e2 0.0,e3 0.0,e4 0.0,e5 0.0,e6 0.0}
DECL FDAT FP643={TOOL_NO 1,BASE_NO 0,IPO_FRAME #BASE}
DECL PDAT PPDAT410={VEL 100.0,ACC 100.0,APO_DIST 100.0}
DECL E6POS XP644={x 1620.0,y -0.00344049511,z 2195.00708,a 0.0,b 89.9996338,c 0.000121682599,s 2,t 34,e1 0.0,e2 0.0,e3 0.0,e4 0.0,e5 0.0,e6 0.0}
DECL FDAT FP644={TOOL_NO 1,BASE_NO 0,IPO_FRAME #BASE}
DECL PDAT PPDAT411={VEL 100.0,ACC 100.0,APO_DIST 100.0}
DECL E6POS XP645={x 1967.90698,y 1049.32898,z 1551.79395,a -152.985992,b 3.54106212,c 173.555695,s 2,t 43,e1 0.0,e2 0.0,e3 0.0,e4 0.0,e5 0.0,e6 0.0}
DECL FDAT FP645={TOOL_NO 1,BASE_NO 0,IPO_FRAME #BASE}
DECL PDAT PPDAT412={VEL 100.0,ACC 100.0,APO_DIST 100.0}
DECL E6POS XP646={x 1887.80298,y 883.617126,z 1660.85498,a -29.7710209,b 34.1978493,c -85.8632202,s 6,t 19,e1 0.0,e2 0.0,e3 0.0,e4 0.0,e5 0.0,e6 0.0}
DECL FDAT FP646={TOOL_NO 1,BASE_NO 0,IPO_FRAME #BASE}
DECL PDAT PPDAT413={VEL 100.0,ACC 100.0,APO_DIST 100.0}
DECL E6POS XP647={x 1887.83398,y 1004.90302,z 1495.27405,a -33.9738503,b 37.2196312,c -84.4143524,s 6,t 19,e1 0.0,e2 0.0,e3 0.0,e4 0.0,e5 0.0,e6 0.0}
DECL FDAT FP647={TOOL_NO 1,BASE_NO 0,IPO_FRAME #BASE}
DECL PDAT PPDAT414={VEL 100.0,ACC 100.0,APO_DIST 100.0}
DECL E6POS XP648={x 1887.83704,y 1017.87598,z 1512.09998,a -33.9738007,b 37.2195892,c -84.4141922,s 6,t 19,e1 0.0,e2 0.0,e3 0.0,e4 0.0,e5 0.0,e6 0.0}
DECL FDAT FP648={TOOL_NO 1,BASE_NO 0,IPO_FRAME #BASE}
DECL PDAT PPDAT415={VEL 100.0,ACC 100.0,APO_DIST 100.0}
DECL E6POS XP649={x 1833.88501,y 478.882996,z 2250.78589,a -33.9730911,b 37.2190704,c -84.4153671,s 6,t 51,e1 0.0,e2 0.0,e3 0.0,e4 0.0,e5 0.0,e6 0.0}
DECL FDAT FP649={TOOL_NO 1,BASE_NO 0,IPO_FRAME #BASE}
DECL PDAT PPDAT416={VEL 100.0,ACC 100.0,APO_DIST 100.0}
DECL E6POS XP650={x 1833.59399,y -493.009491,z 2501.44507,a -33.9630699,b 37.1929092,c -84.3842087,s 6,t 50,e1 0.0,e2 0.0,e3 0.0,e4 0.0,e5 0.0,e6 0.0}
DECL FDAT FP650={TOOL_NO 1,BASE_NO 0,IPO_FRAME #BASE}
DECL PDAT PPDAT417={VEL 100.0,ACC 100.0,APO_DIST 100.0}
DECL E6POS XP651={x 1382.573,y -1385.85095,z 2459.28198,a -63.0737991,b 38.8434601,c -84.7276764,s 6,t 50,e1 0.0,e2 0.0,e3 0.0,e4 0.0,e5 0.0,e6 0.0}
DECL FDAT FP651={TOOL_NO 1,BASE_NO 0,IPO_FRAME #BASE}
DECL PDAT PPDAT418={VEL 100.0,ACC 100.0,APO_DIST 100.0}
DECL E6POS XP652={x 1676.92004,y -1772.95898,z 1712.31396,a -68.0946274,b 32.2391891,c -92.3445969,s 6,t 50,e1 0.0,e2 0.0,e3 0.0,e4 0.0,e5 0.0,e6 0.0}
DECL FDAT FP652={TOOL_NO 1,BASE_NO 0,IPO_FRAME #BASE}
DECL PDAT PPDAT419={VEL 100.0,ACC 100.0,APO_DIST 100.0}
DECL E6POS XP653={x -1259.39697,y 56.1642494,z 1821.02795,a 22.2459602,b 3.90171003,c -178.198502,s 2,t 2,e1 0.0,e2 0.0,e3 0.0,e4 0.0,e5 0.0,e6 0.0}
DECL FDAT FP653={TOOL_NO 1,BASE_NO 0,IPO_FRAME #BASE}
DECL PDAT PPDAT420={VEL 100.0,ACC 100.0,APO_DIST 100.0}
DECL E6POS XP654={x -0.00784905441,y -1260.64502,z 1821.02405,a 114.799103,b 3.90148902,c -178.198593,s 2,t 2,e1 0.0,e2 0.0,e3 0.0,e4 0.0,e5 0.0,e6 0.0}
DECL FDAT FP654={TOOL_NO 1,BASE_NO 0,IPO_FRAME #BASE}
DECL PDAT PPDAT421={VEL 100.0,ACC 100.0,APO_DIST 100.0}
DECL E6POS XP655={x 1260.646,y -0.0358363688,z 1821.02295,a -155.202103,b 3.90116596,c -178.198593,s 2,t 2,e1 0.0,e2 0.0,e3 0.0,e4 0.0,e5 0.0,e6 0.0}
DECL FDAT FP655={TOOL_NO 1,BASE_NO 0,IPO_FRAME #BASE}
DECL PDAT PPDAT422={VEL 100.0,ACC 100.0,APO_DIST 100.0}
DECL E6POS XP656={x 178.423798,y 1247.953,z 1821.02197,a -73.3368835,b 3.90115809,c -178.198593,s 2,t 3,e1 0.0,e2 0.0,e3 0.0,e4 0.0,e5 0.0,e6 0.0}
DECL FDAT FP656={TOOL_NO 1,BASE_NO 0,IPO_FRAME #BASE}
DECL PDAT PPDAT423={VEL 100.0,ACC 100.0,APO_DIST 100.0}
DECL E6POS XP657={x 185.366394,y 1296.51294,z 2275.04199,a -69.4081573,b 29.4691601,c -164.908096,s 2,t 3,e1 0.0,e2 0.0,e3 0.0,e4 0.0,e5 0.0,e6 0.0}
DECL FDAT FP657={TOOL_NO 1,BASE_NO 0,IPO_FRAME #BASE}
DECL PDAT PPDAT424={VEL 100.0,ACC 100.0,APO_DIST 100.0}
DECL E6POS XP658={x -1309.61304,y 15.3324299,z 2275.03296,a 28.0574207,b 29.4685593,c -164.908707,s 2,t 3,e1 0.0,e2 0.0,e3 0.0,e4 0.0,e5 0.0,e6 0.0}
DECL FDAT FP658={TOOL_NO 1,BASE_NO 0,IPO_FRAME #BASE}
DECL PDAT PPDAT425={VEL 100.0,ACC 100.0,APO_DIST 100.0}
DECL E6POS XP659={x 1309.70398,y -0.0697228834,z 2275.021,a -151.275101,b 29.4677792,c -164.909103,s 2,t 2,e1 0.0,e2 0.0,e3 0.0,e4 0.0,e5 0.0,e6 0.0}
DECL FDAT FP659={TOOL_NO 1,BASE_NO 0,IPO_FRAME #BASE}
DECL PDAT PPDAT426={VEL 100.0,ACC 100.0,APO_DIST 100.0}
DECL E6POS XP660={x 494.486786,y -0.0271208696,z 2508.83398,a -132.296295,b 55.5475388,c -137.809402,s 2,t 2,e1 0.0,e2 0.0,e3 0.0,e4 0.0,e5 0.0,e6 0.0}
DECL FDAT FP660={TOOL_NO 1,BASE_NO 0,IPO_FRAME #BASE}
DECL PDAT PPDAT427={VEL 100.0,ACC 100.0,APO_DIST 100.0}
DECL E6POS XP661={x 2769.32495,y -0.129079506,z 1090.15295,a -79.870163,b 64.8421631,c -78.831131,s 4,t 18,e1 0.0,e2 0.0,e3 0.0,e4 0.0,e5 0.0,e6 0.0}
DECL FDAT FP661={TOOL_NO 1,BASE_NO 0,IPO_FRAME #BASE}
DECL PDAT PPDAT428={VEL 100.0,ACC 100.0,APO_DIST 100.0}
DECL E6POS XP662={x 2604.51294,y -6.88281488,z 234.356094,a -84.689682,b 67.0945663,c -82.6785812,s 6,t 24,e1 0.0,e2 0.0,e3 0.0,e4 0.0,e5 0.0,e6 0.0}
DECL FDAT FP662={TOOL_NO 1,BASE_NO 0,IPO_FRAME #BASE}
DECL PDAT PPDAT429={VEL 100.0,ACC 100.0,APO_DIST 100.0}
DECL E6POS XP663={x -924.351074,y -6.71793699,z 1096.38904,a -156.226501,b -16.0039005,c 174.631195,s 5,t 30,e1 0.0,e2 0.0,e3 0.0,e4 0.0,e5 0.0,e6 0.0}
DECL FDAT FP663={TOOL_NO 1,BASE_NO 0,IPO_FRAME #BASE}
DECL PDAT PPDAT430={VEL 100.0,ACC 100.0,APO_DIST 100.0}
DECL E6POS XP664={x -70.0239868,y -0.953113019,z 3155.9541,a -22.4475403,b -5.33677912,c 2.41968608,s 7,t 26,e1 0.0,e2 0.0,e3 0.0,e4 0.0,e5 0.0,e6 0.0}
DECL FDAT FP664={TOOL_NO 1,BASE_NO 0,IPO_FRAME #BASE}
DECL PDAT PPDAT431={VEL 100.0,ACC 100.0,APO_DIST 100.0}
DECL E6POS XP665={x -275.734314,y 66.0350189,z 2768.47607,a 30.8886509,b 54.4333611,c -139.203598,s 3,t 2,e1 0.0,e2 0.0,e3 0.0,e4 0.0,e5 0.0,e6 0.0}
DECL FDAT FP665={TOOL_NO 1,BASE_NO 0,IPO_FRAME #BASE}
DECL PDAT PPDAT432={VEL 100.0,ACC 100.0,APO_DIST 100.0}
DECL E6POS XP666={x -48.7166595,y -0.101860903,z 3157.29297,a -20.6361294,b -1.22956395,c 0.486549199,s 7,t 26,e1 0.0,e2 0.0,e3 0.0,e4 0.0,e5 0.0,e6 0.0}
DECL FDAT FP666={TOOL_NO 1,BASE_NO 0,IPO_FRAME #BASE}
DECL PDAT PPDAT433={VEL 100.0,ACC 100.0,APO_DIST 100.0}
DECL E6POS XP667={x 1886.26794,y -6.82388878,z 1576.46106,a -79.6724014,b 66.2891464,c -77.1833267,s 6,t 26,e1 0.0,e2 0.0,e3 0.0,e4 0.0,e5 0.0,e6 0.0}
DECL FDAT FP667={TOOL_NO 1,BASE_NO 0,IPO_FRAME #BASE}
DECL PDAT PPDAT434={VEL 100.0,ACC 100.0,APO_DIST 100.0}
DECL E6POS XP668={x 2618.34497,y -6.80781603,z 1576.66797,a -79.6421967,b 66.2928391,c -77.154129,s 6,t 26,e1 0.0,e2 0.0,e3 0.0,e4 0.0,e5 0.0,e6 0.0}
DECL FDAT FP668={TOOL_NO 1,BASE_NO 0,IPO_FRAME #BASE}
DECL PDAT PPDAT435={VEL 100.0,ACC 100.0,APO_DIST 100.0}
DECL E6POS XP669={x 1673.44995,y -6.81381893,z 1238.78198,a -79.6456223,b 66.293457,c -77.1576004,s 6,t 26,e1 0.0,e2 0.0,e3 0.0,e4 0.0,e5 0.0,e6 0.0}
DECL FDAT FP669={TOOL_NO 1,BASE_NO 0,IPO_FRAME #BASE}
DECL PDAT PPDAT436={VEL 100.0,ACC 100.0,APO_DIST 100.0}
DECL E6POS XP670={x 1673.50403,y 1954.27405,z 1238.80505,a -79.6490631,b 66.2979431,c -77.1584091,s 6,t 27,e1 0.0,e2 0.0,e3 0.0,e4 0.0,e5 0.0,e6 0.0}
DECL FDAT FP670={TOOL_NO 1,BASE_NO 0,IPO_FRAME #BASE}
DECL PDAT PPDAT437={VEL 100.0,ACC 100.0,APO_DIST 100.0}
DECL E6POS XP671={x 1562.32996,y 212.674103,z 2066.0481,a -79.679863,b 66.3107376,c -77.1943665,s 6,t 27,e1 0.0,e2 0.0,e3 0.0,e4 0.0,e5 0.0,e6 0.0}
DECL FDAT FP671={TOOL_NO 1,BASE_NO 0,IPO_FRAME #BASE}
DECL PDAT PPDAT438={VEL 100.0,ACC 100.0,APO_DIST 100.0}
DECL E6POS XP672={x 1562.22095,y 212.721497,z 2066.03003,a -170.397095,b 66.3151932,c -77.1821518,s 6,t 27,e1 0.0,e2 0.0,e3 0.0,e4 0.0,e5 0.0,e6 0.0}
DECL FDAT FP672={TOOL_NO 1,BASE_NO 0,IPO_FRAME #BASE}
DECL PDAT PPDAT439={VEL 100.0,ACC 100.0,APO_DIST 100.0}
DECL E6POS XP673={x 1562.20496,y 212.482193,z 2066.13403,a -131.142502,b -40.623291,c -6.48490477,s 6,t 27,e1 0.0,e2 0.0,e3 0.0,e4 0.0,e5 0.0,e6 0.0}
DECL FDAT FP673={TOOL_NO 1,BASE_NO 0,IPO_FRAME #BASE}
DECL PDAT PPDAT440={VEL 100.0,ACC 100.0,APO_DIST 100.0}
DECL E6POS XP674={x 1561.974,y 212.410797,z 2965.177,a -131.1754,b -40.6134911,c -6.46997213,s 6,t 27,e1 0.0,e2 0.0,e3 0.0,e4 0.0,e5 0.0,e6 0.0}
DECL FDAT FP674={TOOL_NO 1,BASE_NO 0,IPO_FRAME #BASE}
DECL PDAT PPDAT441={VEL 100.0,ACC 100.0,APO_DIST 100.0}
DECL E6POS XP675={x -735.696289,y -1023.72101,z 1821.02502,a 79.0965424,b 3.90134406,c -178.1987,s 2,t 2,e1 0.0,e2 0.0,e3 0.0,e4 0.0,e5 0.0,e6 0.0}
DECL FDAT FP675={TOOL_NO 1,BASE_NO 0,IPO_FRAME #BASE}
DECL PDAT PPDAT442={VEL 100.0,ACC 100.0,APO_DIST 100.0}
DECL E6POS XP676={x -1239.31604,y -1420.88696,z 650.053223,a 79.0959396,b 3.9004271,c -178.199203,s 2,t 10,e1 0.0,e2 0.0,e3 0.0,e4 0.0,e5 0.0,e6 0.0}
DECL FDAT FP676={TOOL_NO 1,BASE_NO 0,IPO_FRAME #BASE}
DECL PDAT PPDAT443={VEL 100.0,ACC 100.0,APO_DIST 100.0}
DECL E6POS XP677={x -1737.84204,y -1420.88501,z 663.574585,a 79.096138,b 3.90031505,c -178.199295,s 2,t 10,e1 0.0,e2 0.0,e3 0.0,e4 0.0,e5 0.0,e6 0.0}
DECL FDAT FP677={TOOL_NO 1,BASE_NO 0,IPO_FRAME #BASE}
DECL PDAT PPDAT444={VEL 100.0,ACC 100.0,APO_DIST 100.0}
DECL E6POS XP678={x -884.529175,y -1420.88403,z 903.396423,a 79.0961533,b 3.900563,c -178.199295,s 2,t 2,e1 0.0,e2 0.0,e3 0.0,e4 0.0,e5 0.0,e6 0.0}
DECL FDAT FP678={TOOL_NO 1,BASE_NO 0,IPO_FRAME #BASE}
DECL PDAT PPDAT445={VEL 100.0,ACC 100.0,APO_DIST 100.0}
DECL E6POS XP679={x -791.202576,y -1420.89502,z 474.415985,a 93.4293518,b 11.0712099,c -90.3091125,s 2,t 34,e1 0.0,e2 0.0,e3 0.0,e4 0.0,e5 0.0,e6 0.0}
DECL FDAT FP679={TOOL_NO 1,BASE_NO 0,IPO_FRAME #BASE}
DECL PDAT PPDAT446={VEL 100.0,ACC 100.0,APO_DIST 100.0}
DECL E6POS XP680={x -1006.53601,y -1420.89099,z 474.412598,a 93.4295731,b 11.0708799,c -90.3092117,s 2,t 34,e1 0.0,e2 0.0,e3 0.0,e4 0.0,e5 0.0,e6 0.0}
DECL FDAT FP680={TOOL_NO 1,BASE_NO 0,IPO_FRAME #BASE}
DECL PDAT PPDAT447={VEL 100.0,ACC 100.0,APO_DIST 100.0}
DECL E6POS XP681={x -1006.53699,y -737.253723,z 2537.56592,a 93.4313431,b 11.0746603,c -90.306778,s 2,t 2,e1 0.0,e2 0.0,e3 0.0,e4 0.0,e5 0.0,e6 0.0}
DECL FDAT FP681={TOOL_NO 1,BASE_NO 0,IPO_FRAME #BASE}
DECL PDAT PPDAT448={VEL 100.0,ACC 100.0,APO_DIST 100.0}
DECL E6POS XP682={x -1281.27405,y -517.797485,z 3032.66309,a 101.356102,b 1.88191795,c -0.331912786,s 2,t 34,e1 0.0,e2 0.0,e3 0.0,e4 0.0,e5 0.0,e6 0.0}
DECL FDAT FP682={TOOL_NO 1,BASE_NO 0,IPO_FRAME #BASE}
DECL PDAT PPDAT449={VEL 100.0,ACC 100.0,APO_DIST 100.0}
DECL E6POS XP683={x -1011.58502,y -517.720276,z 3115.49707,a 101.358498,b 1.882321,c -0.324090987,s 2,t 34,e1 0.0,e2 0.0,e3 0.0,e4 0.0,e5 0.0,e6 0.0}
DECL FDAT FP683={TOOL_NO 1,BASE_NO 0,IPO_FRAME #BASE}
DECL PDAT PPDAT450={VEL 100.0,ACC 100.0,APO_DIST 100.0}
DECL E6POS XP684={x -1248.96802,y -156.828903,z 2223.06299,a -167.198105,b 79.0125809,c 103.242996,s 2,t 34,e1 0.0,e2 0.0,e3 0.0,e4 0.0,e5 0.0,e6 0.0}
DECL FDAT FP684={TOOL_NO 1,BASE_NO 0,IPO_FRAME #BASE}
DECL PDAT PPDAT451={VEL 100.0,ACC 100.0,APO_DIST 100.0}
DECL E6POS XP685={x -1689.27002,y -156.835007,z 1986.20605,a -167.199097,b 79.012207,c 103.242104,s 2,t 34,e1 0.0,e2 0.0,e3 0.0,e4 0.0,e5 0.0,e6 0.0}
DECL FDAT FP685={TOOL_NO 1,BASE_NO 0,IPO_FRAME #BASE}
DECL PDAT PPDAT452={VEL 100.0,ACC 100.0,APO_DIST 100.0}
DECL E6POS XP686={x -1689.27502,y 93.621048,z 1986.20105,a -167.198395,b 79.0123367,c 103.2425,s 2,t 34,e1 0.0,e2 0.0,e3 0.0,e4 0.0,e5 0.0,e6 0.0}
DECL FDAT FP686={TOOL_NO 1,BASE_NO 0,IPO_FRAME #BASE}
DECL PDAT PPDAT453={VEL 100.0,ACC 100.0,APO_DIST 100.0}
DECL E6POS XP687={x -1689.27295,y -106.853699,z 1986.19495,a -167.198898,b 79.0132065,c 103.241997,s 2,t 34,e1 0.0,e2 0.0,e3 0.0,e4 0.0,e5 0.0,e6 0.0}
DECL FDAT FP687={TOOL_NO 1,BASE_NO 0,IPO_FRAME #BASE}
DECL PDAT PPDAT454={VEL 100.0,ACC 100.0,APO_DIST 100.0}
DECL E6POS XP688={x -1688.625,y -106.8694,z 2441.01001,a -167.188797,b 79.0096207,c 103.253502,s 2,t 34,e1 0.0,e2 0.0,e3 0.0,e4 0.0,e5 0.0,e6 0.0}
DECL FDAT FP688={TOOL_NO 1,BASE_NO 0,IPO_FRAME #BASE}
DECL PDAT PPDAT455={VEL 100.0,ACC 100.0,APO_DIST 100.0}
DECL E6POS XP689={x -802.124573,y -107.313103,z 2702.49512,a 97.9455872,b 3.245543,c -0.0722893625,s 2,t 34,e1 0.0,e2 0.0,e3 0.0,e4 0.0,e5 0.0,e6 0.0}
DECL FDAT FP689={TOOL_NO 1,BASE_NO 0,IPO_FRAME #BASE}
DECL PDAT PPDAT456={VEL 100.0,ACC 100.0,APO_DIST 100.0}
DECL E6POS XP690={x -1077.01294,y 57.9976006,z 2447.7561,a -92.7304993,b 0.737935603,c 86.8507767,s 2,t 42,e1 0.0,e2 0.0,e3 0.0,e4 0.0,e5 0.0,e6 0.0}
DECL FDAT FP690={TOOL_NO 1,BASE_NO 0,IPO_FRAME #BASE}
DECL PDAT PPDAT457={VEL 100.0,ACC 100.0,APO_DIST 100.0}
DECL E6POS XP691={x -1268.34094,y 67.2796707,z 2370.57397,a -91.8260269,b 0.675085783,c 85.2613068,s 2,t 42,e1 0.0,e2 0.0,e3 0.0,e4 0.0,e5 0.0,e6 0.0}
DECL FDAT FP691={TOOL_NO 1,BASE_NO 0,IPO_FRAME #BASE}
DECL PDAT PPDAT458={VEL 100.0,ACC 100.0,APO_DIST 100.0}
DECL E6POS XP692={x -1268.34094,y 67.2796707,z 2370.57397,a -91.8260269,b 0.675085783,c 85.2613068,s 2,t 42,e1 0.0,e2 0.0,e3 0.0,e4 0.0,e5 0.0,e6 0.0}
DECL FDAT FP692={TOOL_NO 1,BASE_NO 0,IPO_FRAME #BASE}
DECL LDAT LCPDAT204={VEL 2.0,ACC 100.0,APO_DIST 100.0,APO_FAC 50.0}
DECL E6POS XP693={x -1383.86694,y 95.9401627,z 1186.88599,a -94.6206589,b 7.83129787,c 86.1557388,s 6,t 58,e1 0.0,e2 0.0,e3 0.0,e4 0.0,e5 0.0,e6 0.0}
DECL FDAT FP693={TOOL_NO 1,BASE_NO 0,IPO_FRAME #BASE}
DECL PDAT PPDAT459={VEL 100.0,ACC 100.0,APO_DIST 100.0}
DECL E6POS XP694={x 2433.47705,y 442.98941,z 1132.82495,a 179.476105,b 4.27273703,c 176.887604,s 2,t 43,e1 0.0,e2 0.0,e3 0.0,e4 0.0,e5 0.0,e6 0.0}
DECL FDAT FP694={TOOL_NO 1,BASE_NO 0,IPO_FRAME #BASE}
DECL PDAT PPDAT460={VEL 100.0,ACC 100.0,APO_DIST 100.0}
DECL E6POS XP695={x 2433.46802,y 442.991608,z 578.324829,a 179.476196,b 4.27178383,c 176.888107,s 2,t 43,e1 0.0,e2 0.0,e3 0.0,e4 0.0,e5 0.0,e6 0.0}
DECL FDAT FP695={TOOL_NO 1,BASE_NO 0,IPO_FRAME #BASE}
DECL PDAT PPDAT461={VEL 100.0,ACC 100.0,APO_DIST 100.0}
DECL E6POS XP696={x 2433.47095,y 442.993195,z 712.214783,a 179.476395,b 4.27213478,c 176.887802,s 2,t 43,e1 0.0,e2 0.0,e3 0.0,e4 0.0,e5 0.0,e6 0.0}
DECL FDAT FP696={TOOL_NO 1,BASE_NO 0,IPO_FRAME #BASE}
DECL PDAT PPDAT462={VEL 100.0,ACC 100.0,APO_DIST 100.0}
DECL E6POS XP697={x 344.546387,y 363.753693,z 3173.65894,a 33.5704803,b 39.4743614,c -10.7840004,s 2,t 11,e1 0.0,e2 0.0,e3 0.0,e4 0.0,e5 0.0,e6 0.0}
DECL FDAT FP697={TOOL_NO 1,BASE_NO 0,IPO_FRAME #BASE}
DECL PDAT PPDAT463={VEL 100.0,ACC 100.0,APO_DIST 100.0}
DECL E6POS XP698={x -588.510071,y -637.426208,z 1952.93506,a -120.657898,b 3.31128407,c -177.518494,s 5,t 31,e1 0.0,e2 0.0,e3 0.0,e4 0.0,e5 0.0,e6 0.0}
DECL FDAT FP698={TOOL_NO 1,BASE_NO 0,IPO_FRAME #BASE}
DECL PDAT PPDAT464={VEL 100.0,ACC 100.0,APO_DIST 100.0}
DECL E6POS XP699={x -588.5047,y -637.421021,z 1101.62,a -120.657501,b 3.31174898,c -177.518295,s 5,t 31,e1 0.0,e2 0.0,e3 0.0,e4 0.0,e5 0.0,e6 0.0}
DECL FDAT FP699={TOOL_NO 1,BASE_NO 0,IPO_FRAME #BASE}
DECL PDAT PPDAT465={VEL 100.0,ACC 100.0,APO_DIST 100.0}
DECL E6POS XP700={x -588.501526,y -637.420105,z 1975.38501,a -120.6576,b 3.31102705,c -177.518494,s 5,t 31,e1 0.0,e2 0.0,e3 0.0,e4 0.0,e5 0.0,e6 0.0}
DECL FDAT FP700={TOOL_NO 1,BASE_NO 0,IPO_FRAME #BASE}
DECL PDAT PPDAT466={VEL 100.0,ACC 100.0,APO_DIST 100.0}
DECL E6POS XP701={x 961.806702,y 1595.98206,z 2099.47412,a -127.544701,b 4.22827387,c 178.259598,s 2,t 43,e1 0.0,e2 0.0,e3 0.0,e4 0.0,e5 0.0,e6 0.0}
DECL FDAT FP701={TOOL_NO 1,BASE_NO 0,IPO_FRAME #BASE}
DECL PDAT PPDAT467={VEL 100.0,ACC 100.0,APO_DIST 100.0}
DECL E6POS XP702={x 961.809875,y 1595.979,z 1170.96899,a -127.544403,b 4.22824621,c 178.259796,s 2,t 43,e1 0.0,e2 0.0,e3 0.0,e4 0.0,e5 0.0,e6 0.0}
DECL FDAT FP702={TOOL_NO 1,BASE_NO 0,IPO_FRAME #BASE}
DECL PDAT PPDAT468={VEL 100.0,ACC 100.0,APO_DIST 100.0}
DECL E6POS XP703={x 961.807617,y 1595.98096,z 2017.58606,a -127.543701,b 4.22771311,c 178.260101,s 2,t 43,e1 0.0,e2 0.0,e3 0.0,e4 0.0,e5 0.0,e6 0.0}
DECL FDAT FP703={TOOL_NO 1,BASE_NO 0,IPO_FRAME #BASE}
DECL PDAT PPDAT469={VEL 100.0,ACC 100.0,APO_DIST 100.0}
DECL E6POS XP704={x 1617.73706,y -94.3353271,z 2242.49707,a -123.820801,b 2.00038695,c -177.729996,s 2,t 10,e1 0.0,e2 0.0,e3 0.0,e4 0.0,e5 0.0,e6 0.0}
DECL FDAT FP704={TOOL_NO 1,BASE_NO 0,IPO_FRAME #BASE}
DECL PDAT PPDAT470={VEL 100.0,ACC 100.0,APO_DIST 100.0}
DECL E6POS XP705={x 1617.73804,y -94.3381729,z 1538.68005,a -123.820503,b 2.00033307,c -177.730301,s 2,t 10,e1 0.0,e2 0.0,e3 0.0,e4 0.0,e5 0.0,e6 0.0}
DECL FDAT FP705={TOOL_NO 1,BASE_NO 0,IPO_FRAME #BASE}
DECL PDAT PPDAT471={VEL 100.0,ACC 100.0,APO_DIST 100.0}
DECL E6POS XP706={x 1617.74597,y -94.3351212,z 678.250916,a -123.820198,b 2.00053,c -177.729996,s 2,t 10,e1 0.0,e2 0.0,e3 0.0,e4 0.0,e5 0.0,e6 0.0}
DECL FDAT FP706={TOOL_NO 1,BASE_NO 0,IPO_FRAME #BASE}
DECL PDAT PPDAT472={VEL 100.0,ACC 100.0,APO_DIST 100.0}
DECL E6POS XP707={x 1617.677,y -94.3300705,z 563.035278,a -123.825401,b 1.99857497,c -177.734299,s 2,t 10,e1 0.0,e2 0.0,e3 0.0,e4 0.0,e5 0.0,e6 0.0}
DECL FDAT FP707={TOOL_NO 1,BASE_NO 0,IPO_FRAME #BASE}
DECL PDAT PPDAT473={VEL 100.0,ACC 100.0,APO_DIST 100.0}
DECL E6POS XP708={x 1617.66504,y -94.3295364,z 655.982483,a -123.825203,b 1.99756205,c -177.735901,s 2,t 10,e1 0.0,e2 0.0,e3 0.0,e4 0.0,e5 0.0,e6 0.0}
DECL FDAT FP708={TOOL_NO 1,BASE_NO 0,IPO_FRAME #BASE}
DECL PDAT PPDAT474={VEL 100.0,ACC 100.0,APO_DIST 100.0}
DECL E6POS XP709={x 1619.99805,y -0.00344048999,z 1549.68201,a -89.9992371,b 65.9794464,c -89.9990311,s 6,t 18,e1 0.0,e2 0.0,e3 0.0,e4 0.0,e5 0.0,e6 0.0}
DECL FDAT FP709={TOOL_NO 1,BASE_NO 0,IPO_FRAME #BASE}
DECL PDAT PPDAT475={VEL 100.0,ACC 100.0,APO_DIST 100.0}
DECL E6POS XP710={x 1298.31799,y 870.844788,z 1480.88098,a -153.193604,b -0.451602399,c 175.890106,s 6,t 27,e1 0.0,e2 0.0,e3 0.0,e4 0.0,e5 0.0,e6 0.0}
DECL FDAT FP710={TOOL_NO 1,BASE_NO 0,IPO_FRAME #BASE}
DECL PDAT PPDAT476={VEL 100.0,ACC 100.0,APO_DIST 100.0}
DECL E6POS XP711={x 1089.03601,y 911.322083,z 1202.63306,a -153.194107,b 0.692702889,c 176.4655,s 6,t 27,e1 0.0,e2 0.0,e3 0.0,e4 0.0,e5 0.0,e6 0.0}
DECL FDAT FP711={TOOL_NO 1,BASE_NO 0,IPO_FRAME #BASE}
DECL PDAT PPDAT477={VEL 100.0,ACC 100.0,APO_DIST 100.0}
DECL E6POS XP712={x 1685.75098,y 418.688507,z 461.656189,a -153.204407,b 0.690404117,c 176.461594,s 6,t 27,e1 0.0,e2 0.0,e3 0.0,e4 0.0,e5 0.0,e6 0.0}
DECL FDAT FP712={TOOL_NO 1,BASE_NO 0,IPO_FRAME #BASE}
DECL PDAT PPDAT478={VEL 100.0,ACC 100.0,APO_DIST 100.0}
DECL E6POS XP713={x 1685.75098,y 418.688507,z 461.656189,a -153.204407,b 0.690404117,c 176.461594,s 6,t 27,e1 0.0,e2 0.0,e3 0.0,e4 0.0,e5 0.0,e6 0.0}
DECL FDAT FP713={TOOL_NO 1,BASE_NO 0,IPO_FRAME #BASE}
DECL LDAT LCPDAT205={VEL 2.0,ACC 100.0,APO_DIST 100.0,APO_FAC 50.0}
DECL E6POS XP714={x 2119.49292,y 418.76889,z 442.606903,a -153.201797,b 0.692657113,c 176.461105,s 6,t 27,e1 0.0,e2 0.0,e3 0.0,e4 0.0,e5 0.0,e6 0.0}
DECL FDAT FP714={TOOL_NO 1,BASE_NO 0,IPO_FRAME #BASE}
DECL LDAT LCPDAT206={VEL 2.0,ACC 100.0,APO_DIST 100.0,APO_FAC 50.0}
DECL E6POS XP715={x 2119.50098,y 418.770996,z 1339.03699,a -153.201706,b 0.693627,c 176.461304,s 6,t 27,e1 0.0,e2 0.0,e3 0.0,e4 0.0,e5 0.0,e6 0.0}
DECL FDAT FP715={TOOL_NO 1,BASE_NO 0,IPO_FRAME #BASE}
DECL LDAT LCPDAT207={VEL 2.0,ACC 100.0,APO_DIST 100.0,APO_FAC 50.0}
DECL E6POS XP716={x 1354.71997,y -6.99321795,z 1800.33301,a -171.503098,b 0.6939556,c 176.461197,s 6,t 26,e1 0.0,e2 0.0,e3 0.0,e4 0.0,e5 0.0,e6 0.0}
DECL FDAT FP716={TOOL_NO 1,BASE_NO 0,IPO_FRAME #BASE}
DECL PDAT PPDAT479={VEL 100.0,ACC 100.0,APO_DIST 100.0}
DECL E6POS XP717={x -166.082199,y -1353.85095,z 1225.04797,a -115.924103,b 1.32480097,c -176.645996,s 6,t 26,e1 0.0,e2 0.0,e3 0.0,e4 0.0,e5 0.0,e6 0.0}
DECL FDAT FP717={TOOL_NO 1,BASE_NO 0,IPO_FRAME #BASE}
DECL PDAT PPDAT480={VEL 100.0,ACC 100.0,APO_DIST 100.0}
DECL E6POS XP718={x -1486.64697,y -1353.79797,z 1175.16003,a 27.0150604,b -3.07961798,c 178.120407,s 6,t 26,e1 0.0,e2 0.0,e3 0.0,e4 0.0,e5 0.0,e6 0.0}
DECL FDAT FP718={TOOL_NO 1,BASE_NO 0,IPO_FRAME #BASE}
DECL PDAT PPDAT481={VEL 100.0,ACC 100.0,APO_DIST 100.0}
DECL E6POS XP719={x -1486.64697,y -1353.79895,z 1088.72095,a 27.0151405,b -3.07967401,c 178.120407,s 6,t 26,e1 0.0,e2 0.0,e3 0.0,e4 0.0,e5 0.0,e6 0.0}
DECL FDAT FP719={TOOL_NO 1,BASE_NO 0,IPO_FRAME #BASE}
DECL PDAT PPDAT482={VEL 100.0,ACC 100.0,APO_DIST 100.0}
DECL E6POS XP720={x -1205.68103,y -1353.79895,z 1088.724,a 27.0152798,b -3.07954788,c 178.1203,s 6,t 26,e1 0.0,e2 0.0,e3 0.0,e4 0.0,e5 0.0,e6 0.0}
DECL FDAT FP720={TOOL_NO 1,BASE_NO 0,IPO_FRAME #BASE}
DECL PDAT PPDAT483={VEL 100.0,ACC 100.0,APO_DIST 100.0}
DECL E6POS XP721={x -657.08728,y -1353.80005,z 1072.39697,a 27.0152206,b -3.07920194,c 178.120193,s 6,t 26,e1 0.0,e2 0.0,e3 0.0,e4 0.0,e5 0.0,e6 0.0}
DECL FDAT FP721={TOOL_NO 1,BASE_NO 0,IPO_FRAME #BASE}
DECL PDAT PPDAT484={VEL 100.0,ACC 100.0,APO_DIST 100.0}
DECL E6POS XP722={x 771.930298,y 1505.81897,z 1209.23999,a -152.936401,b -0.383393586,c 177.852905,s 6,t 27,e1 0.0,e2 0.0,e3 0.0,e4 0.0,e5 0.0,e6 0.0}
DECL FDAT FP722={TOOL_NO 1,BASE_NO 0,IPO_FRAME #BASE}
DECL PDAT PPDAT485={VEL 100.0,ACC 100.0,APO_DIST 100.0}
DECL E6POS XP723={x 1592.32495,y 1505.82104,z 1209.23706,a -152.936096,b -0.383576512,c 177.852798,s 6,t 27,e1 0.0,e2 0.0,e3 0.0,e4 0.0,e5 0.0,e6 0.0}
DECL FDAT FP723={TOOL_NO 1,BASE_NO 0,IPO_FRAME #BASE}
DECL PDAT PPDAT486={VEL 100.0,ACC 100.0,APO_DIST 100.0}
DECL E6POS XP724={x 1592.32495,y 1505.82104,z 1209.23706,a -152.936096,b -0.383576512,c 177.852798,s 6,t 27,e1 0.0,e2 0.0,e3 0.0,e4 0.0,e5 0.0,e6 0.0}
DECL FDAT FP724={TOOL_NO 1,BASE_NO 0,IPO_FRAME #BASE}
DECL LDAT LCPDAT208={VEL 2.0,ACC 100.0,APO_DIST 100.0,APO_FAC 50.0}
DECL E6POS XP725={x 1797.73303,y 1506.22205,z 1209.85303,a -152.967697,b -0.351146102,c 177.841995,s 6,t 27,e1 0.0,e2 0.0,e3 0.0,e4 0.0,e5 0.0,e6 0.0}
DECL FDAT FP725={TOOL_NO 1,BASE_NO 0,IPO_FRAME #BASE}
DECL LDAT LCPDAT209={VEL 2.0,ACC 100.0,APO_DIST 100.0,APO_FAC 50.0}
DECL E6POS XP726={x 1797.73499,y 1506.21704,z 1299.35498,a -152.967804,b -0.351565897,c 177.842102,s 6,t 27,e1 0.0,e2 0.0,e3 0.0,e4 0.0,e5 0.0,e6 0.0}
DECL FDAT FP726={TOOL_NO 1,BASE_NO 0,IPO_FRAME #BASE}
DECL LDAT LCPDAT210={VEL 2.0,ACC 100.0,APO_DIST 100.0,APO_FAC 50.0}
DECL E6POS XP727={x 1551.21704,y 1506.20898,z 1299.35706,a -152.967606,b -0.351818413,c 177.841995,s 6,t 27,e1 0.0,e2 0.0,e3 0.0,e4 0.0,e5 0.0,e6 0.0}
DECL FDAT FP727={TOOL_NO 1,BASE_NO 0,IPO_FRAME #BASE}
DECL PDAT PPDAT487={VEL 100.0,ACC 100.0,APO_DIST 100.0}
DECL E6POS XP728={x 1551.21704,y -257.292999,z 1299.35498,a -152.966995,b -0.35214591,c 177.841904,s 6,t 26,e1 0.0,e2 0.0,e3 0.0,e4 0.0,e5 0.0,e6 0.0}
DECL FDAT FP728={TOOL_NO 1,BASE_NO 0,IPO_FRAME #BASE}
DECL PDAT PPDAT488={VEL 100.0,ACC 100.0,APO_DIST 100.0}
DECL E6POS XP729={x 1551.22205,y -1046.38904,z 1299.35901,a 116.517799,b -2.15416908,c -179.629303,s 6,t 26,e1 0.0,e2 0.0,e3 0.0,e4 0.0,e5 0.0,e6 0.0}
DECL FDAT FP729={TOOL_NO 1,BASE_NO 0,IPO_FRAME #BASE}
DECL PDAT PPDAT489={VEL 100.0,ACC 100.0,APO_DIST 100.0}
DECL E6POS XP730={x -1570.94397,y -1046.39502,z 1299.37402,a 116.517799,b -2.15412498,c -179.628296,s 6,t 26,e1 0.0,e2 0.0,e3 0.0,e4 0.0,e5 0.0,e6 0.0}
DECL FDAT FP730={TOOL_NO 1,BASE_NO 0,IPO_FRAME #BASE}
DECL PDAT PPDAT490={VEL 100.0,ACC 100.0,APO_DIST 100.0}
DECL E6POS XP731={x -1570.94897,y -1046.39795,z 1099.44397,a 116.5177,b -2.15415192,c -179.628006,s 6,t 26,e1 0.0,e2 0.0,e3 0.0,e4 0.0,e5 0.0,e6 0.0}
DECL FDAT FP731={TOOL_NO 1,BASE_NO 0,IPO_FRAME #BASE}
DECL PDAT PPDAT491={VEL 100.0,ACC 100.0,APO_DIST 100.0}
DECL E6POS XP732={x -1658.15796,y -1046.40601,z 1099.45398,a 116.517899,b -2.15401101,c -179.627197,s 6,t 26,e1 0.0,e2 0.0,e3 0.0,e4 0.0,e5 0.0,e6 0.0}
DECL FDAT FP732={TOOL_NO 1,BASE_NO 0,IPO_FRAME #BASE}
DECL PDAT PPDAT492={VEL 100.0,ACC 100.0,APO_DIST 100.0}
DECL E6POS XP733={x -1658.15198,y -1046.37598,z 1099.47595,a 114.5765,b 10.7881098,c 151.546402,s 6,t 26,e1 0.0,e2 0.0,e3 0.0,e4 0.0,e5 0.0,e6 0.0}
DECL FDAT FP733={TOOL_NO 1,BASE_NO 0,IPO_FRAME #BASE}
DECL PDAT PPDAT493={VEL 100.0,ACC 100.0,APO_DIST 100.0}
DECL E6POS XP734={x -1658.151,y -1046.38306,z 1245.29297,a 116.489601,b 3.31582689,c 179.461304,s 6,t 26,e1 0.0,e2 0.0,e3 0.0,e4 0.0,e5 0.0,e6 0.0}
DECL FDAT FP734={TOOL_NO 1,BASE_NO 0,IPO_FRAME #BASE}
DECL PDAT PPDAT494={VEL 100.0,ACC 100.0,APO_DIST 100.0}
DECL E6POS XP735={x 2397.41504,y 119.114197,z 1227.48096,a 119.834198,b -2.20159101,c 177.812302,s 6,t 27,e1 0.0,e2 0.0,e3 0.0,e4 0.0,e5 0.0,e6 0.0}
DECL FDAT FP735={TOOL_NO 1,BASE_NO 0,IPO_FRAME #BASE}
DECL PDAT PPDAT495={VEL 100.0,ACC 100.0,APO_DIST 100.0}
DECL E6POS XP736={x 2397.41699,y -193.256195,z 1227.48401,a 119.834099,b -2.20136499,c 177.812103,s 6,t 26,e1 0.0,e2 0.0,e3 0.0,e4 0.0,e5 0.0,e6 0.0}
DECL FDAT FP736={TOOL_NO 1,BASE_NO 0,IPO_FRAME #BASE}
DECL PDAT PPDAT496={VEL 100.0,ACC 100.0,APO_DIST 100.0}
DECL E6POS XP737={x 2397.41699,y -193.256195,z 1227.48401,a 119.834099,b -2.20136499,c 177.812103,s 6,t 26,e1 0.0,e2 0.0,e3 0.0,e4 0.0,e5 0.0,e6 0.0}
DECL FDAT FP737={TOOL_NO 1,BASE_NO 0,IPO_FRAME #BASE}
DECL LDAT LCPDAT211={VEL 2.0,ACC 100.0,APO_DIST 100.0,APO_FAC 50.0}
DECL E6POS XP738={x 2397.41504,y -377.8414,z 1227.47998,a 119.833801,b -2.20167804,c 177.8125,s 6,t 26,e1 0.0,e2 0.0,e3 0.0,e4 0.0,e5 0.0,e6 0.0}
DECL FDAT FP738={TOOL_NO 1,BASE_NO 0,IPO_FRAME #BASE}
DECL LDAT LCPDAT212={VEL 2.0,ACC 100.0,APO_DIST 100.0,APO_FAC 50.0}
DECL E6POS XP739={x 2397.36304,y -377.837799,z 1258.77502,a 119.838303,b -2.20861292,c 177.824402,s 6,t 26,e1 0.0,e2 0.0,e3 0.0,e4 0.0,e5 0.0,e6 0.0}
DECL FDAT FP739={TOOL_NO 1,BASE_NO 0,IPO_FRAME #BASE}
DECL LDAT LCPDAT213={VEL 2.0,ACC 100.0,APO_DIST 100.0,APO_FAC 50.0}
DECL E6POS XP740={x 2397.36499,y 37.3564911,z 1258.78296,a 119.838203,b -2.20832205,c 177.824005,s 6,t 27,e1 0.0,e2 0.0,e3 0.0,e4 0.0,e5 0.0,e6 0.0}
DECL FDAT FP740={TOOL_NO 1,BASE_NO 0,IPO_FRAME #BASE}
DECL PDAT PPDAT497={VEL 100.0,ACC 100.0,APO_DIST 100.0}
DECL E6POS XP741={x 1240.96594,y 1214.224,z 1554.10303,a -150.719894,b 0.70310837,c 179.989105,s 6,t 27,e1 0.0,e2 0.0,e3 0.0,e4 0.0,e5 0.0,e6 0.0}
DECL FDAT FP741={TOOL_NO 1,BASE_NO 0,IPO_FRAME #BASE}
DECL PDAT PPDAT498={VEL 100.0,ACC 100.0,APO_DIST 100.0}
DECL E6POS XP742={x 1651.203,y 1542.56604,z 1326.38904,a 79.3812637,b 1.04392695,c 179.563095,s 6,t 27,e1 0.0,e2 0.0,e3 0.0,e4 0.0,e5 0.0,e6 0.0}
DECL FDAT FP742={TOOL_NO 1,BASE_NO 0,IPO_FRAME #BASE}
DECL PDAT PPDAT499={VEL 100.0,ACC 100.0,APO_DIST 100.0}
DECL E6POS XP743={x 1808.48401,y 1456.40198,z 1268.646,a 79.3529663,b 0.984387517,c 179.520599,s 6,t 27,e1 0.0,e2 0.0,e3 0.0,e4 0.0,e5 0.0,e6 0.0}
DECL FDAT FP743={TOOL_NO 1,BASE_NO 0,IPO_FRAME #BASE}
DECL PDAT PPDAT500={VEL 100.0,ACC 100.0,APO_DIST 100.0}
DECL E6POS XP744={x 691.801025,y 21.2626209,z 1515.44702,a -153.435104,b -4.04898977,c 178.1315,s 2,t 3,e1 0.0,e2 0.0,e3 0.0,e4 0.0,e5 0.0,e6 0.0}
DECL FDAT FP744={TOOL_NO 1,BASE_NO 0,IPO_FRAME #BASE}
DECL PDAT PPDAT501={VEL 100.0,ACC 100.0,APO_DIST 100.0}
DECL E6POS XP745={x 1349.16394,y 172.669205,z 1195.26099,a 117.154602,b 0.838489294,c 175.789307,s 2,t 43,e1 0.0,e2 0.0,e3 0.0,e4 0.0,e5 0.0,e6 0.0}
DECL FDAT FP745={TOOL_NO 1,BASE_NO 0,IPO_FRAME #BASE}
DECL PDAT PPDAT502={VEL 100.0,ACC 100.0,APO_DIST 100.0}
DECL E6POS XP746={x 1349.172,y -58.4891586,z 1195.26794,a 117.154602,b 0.838847518,c 175.788696,s 2,t 42,e1 0.0,e2 0.0,e3 0.0,e4 0.0,e5 0.0,e6 0.0}
DECL FDAT FP746={TOOL_NO 1,BASE_NO 0,IPO_FRAME #BASE}
DECL PDAT PPDAT503={VEL 100.0,ACC 100.0,APO_DIST 100.0}
DECL E6POS XP747={x 1349.172,y -58.4891586,z 1195.26794,a 117.154602,b 0.838847518,c 175.788696,s 2,t 42,e1 0.0,e2 0.0,e3 0.0,e4 0.0,e5 0.0,e6 0.0}
DECL FDAT FP747={TOOL_NO 1,BASE_NO 0,IPO_FRAME #BASE}
DECL LDAT LCPDAT214={VEL 2.0,ACC 100.0,APO_DIST 100.0,APO_FAC 50.0}
DECL E6POS XP748={x 1349.18396,y -218.871597,z 1195.27295,a 117.1549,b 0.839231372,c 175.788193,s 2,t 42,e1 0.0,e2 0.0,e3 0.0,e4 0.0,e5 0.0,e6 0.0}
DECL FDAT FP748={TOOL_NO 1,BASE_NO 0,IPO_FRAME #BASE}
DECL LDAT LCPDAT215={VEL 2.0,ACC 100.0,APO_DIST 100.0,APO_FAC 50.0}
DECL E6POS XP749={x 1349.19897,y -218.873901,z 1238.479,a 117.154701,b 0.839943588,c 175.787201,s 2,t 42,e1 0.0,e2 0.0,e3 0.0,e4 0.0,e5 0.0,e6 0.0}
DECL FDAT FP749={TOOL_NO 1,BASE_NO 0,IPO_FRAME #BASE}
DECL LDAT LCPDAT216={VEL 2.0,ACC 100.0,APO_DIST 100.0,APO_FAC 50.0}
DECL E6POS XP750={x 1349.198,y -218.876205,z 1255.99194,a 117.154099,b 0.840101779,c 175.786697,s 2,t 42,e1 0.0,e2 0.0,e3 0.0,e4 0.0,e5 0.0,e6 0.0}
DECL FDAT FP750={TOOL_NO 1,BASE_NO 0,IPO_FRAME #BASE}
DECL PDAT PPDAT504={VEL 100.0,ACC 100.0,APO_DIST 100.0}
DECL E6POS XP751={x 1349.19202,y 862.53241,z 1417.31299,a 117.154099,b 0.840081811,c 175.787201,s 2,t 35,e1 0.0,e2 0.0,e3 0.0,e4 0.0,e5 0.0,e6 0.0}
DECL FDAT FP751={TOOL_NO 1,BASE_NO 0,IPO_FRAME #BASE}
DECL PDAT PPDAT505={VEL 100.0,ACC 100.0,APO_DIST 100.0}
DECL E6POS XP752={x 1545.40405,y 1556.89502,z 1379.005,a 78.1537933,b -6.88922215,c 179.056702,s 2,t 43,e1 0.0,e2 0.0,e3 0.0,e4 0.0,e5 0.0,e6 0.0}
DECL FDAT FP752={TOOL_NO 1,BASE_NO 0,IPO_FRAME #BASE}
DECL PDAT PPDAT506={VEL 100.0,ACC 100.0,APO_DIST 100.0}
DECL E6POS XP753={x 1545.40198,y 1556.90002,z 1274.64795,a 78.1537399,b -6.88932896,c 179.056595,s 2,t 43,e1 0.0,e2 0.0,e3 0.0,e4 0.0,e5 0.0,e6 0.0}
DECL FDAT FP753={TOOL_NO 1,BASE_NO 0,IPO_FRAME #BASE}
DECL LDAT LCPDAT217={VEL 2.0,ACC 100.0,APO_DIST 100.0,APO_FAC 50.0}
DECL E6POS XP754={x 1545.39697,y 1556.896,z 1210.28003,a 78.1537018,b -6.88900995,c 179.057098,s 2,t 43,e1 0.0,e2 0.0,e3 0.0,e4 0.0,e5 0.0,e6 0.0}
DECL FDAT FP754={TOOL_NO 1,BASE_NO 0,IPO_FRAME #BASE}
DECL LDAT LCPDAT218={VEL 2.0,ACC 100.0,APO_DIST 100.0,APO_FAC 50.0}
DECL E6POS XP755={x 1591.63696,y 1609.74402,z 1210.26099,a 78.1541367,b -6.88918018,c 179.056702,s 2,t 43,e1 0.0,e2 0.0,e3 0.0,e4 0.0,e5 0.0,e6 0.0}
DECL FDAT FP755={TOOL_NO 1,BASE_NO 0,IPO_FRAME #BASE}
DECL PDAT PPDAT507={VEL 100.0,ACC 100.0,APO_DIST 100.0}
DECL E6POS XP756={x 1591.64197,y 1609.74194,z 1487.48096,a 78.1536484,b -6.88963985,c 179.056198,s 2,t 43,e1 0.0,e2 0.0,e3 0.0,e4 0.0,e5 0.0,e6 0.0}
DECL FDAT FP756={TOOL_NO 1,BASE_NO 0,IPO_FRAME #BASE}
DECL PDAT PPDAT508={VEL 100.0,ACC 100.0,APO_DIST 100.0}
DECL E6POS XP757={x 1471.39404,y 1182.349,z 1694.38904,a 78.1538391,b -6.88960505,c 179.056702,s 2,t 43,e1 0.0,e2 0.0,e3 0.0,e4 0.0,e5 0.0,e6 0.0}
DECL FDAT FP757={TOOL_NO 1,BASE_NO 0,IPO_FRAME #BASE}
DECL PDAT PPDAT509={VEL 100.0,ACC 100.0,APO_DIST 100.0}
DECL E6POS XP758={x 1471.39502,y -1333.16602,z 1694.38794,a -60.8894806,b -3.98855209,c -177.020401,s 2,t 10,e1 0.0,e2 0.0,e3 0.0,e4 0.0,e5 0.0,e6 0.0}
DECL FDAT FP758={TOOL_NO 1,BASE_NO 0,IPO_FRAME #BASE}
DECL PDAT PPDAT510={VEL 100.0,ACC 100.0,APO_DIST 100.0}
DECL E6POS XP759={x 1408.41504,y -1349.28296,z 1206.39197,a -63.8400192,b -3.98088002,c -177.018906,s 2,t 10,e1 0.0,e2 0.0,e3 0.0,e4 0.0,e5 0.0,e6 0.0}
DECL FDAT FP759={TOOL_NO 1,BASE_NO 0,IPO_FRAME #BASE}
DECL PDAT PPDAT511={VEL 100.0,ACC 100.0,APO_DIST 100.0}
DECL E6POS XP760={x 1408.41895,y -1346.00195,z 1209.36597,a -63.8400917,b -3.98153496,c -177.018707,s 2,t 10,e1 0.0,e2 0.0,e3 0.0,e4 0.0,e5 0.0,e6 0.0}
DECL FDAT FP760={TOOL_NO 1,BASE_NO 0,IPO_FRAME #BASE}
DECL LDAT LCPDAT219={VEL 2.0,ACC 100.0,APO_DIST 100.0,APO_FAC 50.0}
DECL E6POS XP761={x 1408.40601,y -1080.09094,z 1209.35706,a -63.8404884,b -3.98085308,c -177.018997,s 2,t 10,e1 0.0,e2 0.0,e3 0.0,e4 0.0,e5 0.0,e6 0.0}
DECL FDAT FP761={TOOL_NO 1,BASE_NO 0,IPO_FRAME #BASE}
DECL LDAT LCPDAT220={VEL 2.0,ACC 100.0,APO_DIST 100.0,APO_FAC 50.0}
DECL E6POS XP762={x 1408.401,y -1080.08997,z 1317.82495,a -63.8410683,b -3.98059011,c -177.018799,s 2,t 10,e1 0.0,e2 0.0,e3 0.0,e4 0.0,e5 0.0,e6 0.0}
DECL FDAT FP762={TOOL_NO 1,BASE_NO 0,IPO_FRAME #BASE}
DECL LDAT LCPDAT221={VEL 2.0,ACC 100.0,APO_DIST 100.0,APO_FAC 50.0}
DECL E6POS XP763={x 1408.39294,y -1080.08801,z 1399.44495,a -63.8416786,b -3.98002505,c -177.018906,s 2,t 10,e1 0.0,e2 0.0,e3 0.0,e4 0.0,e5 0.0,e6 0.0}
DECL FDAT FP763={TOOL_NO 1,BASE_NO 0,IPO_FRAME #BASE}
DECL PDAT PPDAT512={VEL 100.0,ACC 100.0,APO_DIST 100.0}
DECL E6POS XP764={x 1408.39905,y 543.555176,z 1556.43298,a -64.1510773,b 2.18950701,c -175.761398,s 2,t 11,e1 0.0,e2 0.0,e3 0.0,e4 0.0,e5 0.0,e6 0.0}
DECL FDAT FP764={TOOL_NO 1,BASE_NO 0,IPO_FRAME #BASE}
DECL PDAT PPDAT513={VEL 100.0,ACC 100.0,APO_DIST 100.0}
DECL E6POS XP765={x 1026.92297,y 887.216675,z 1395.66602,a -104.7341,b 4.24522114,c -178.286896,s 2,t 11,e1 0.0,e2 0.0,e3 0.0,e4 0.0,e5 0.0,e6 0.0}
DECL FDAT FP765={TOOL_NO 1,BASE_NO 0,IPO_FRAME #BASE}
DECL PDAT PPDAT514={VEL 100.0,ACC 100.0,APO_DIST 100.0}
DECL E6POS XP766={x 1026.922,y 887.215698,z 1261.52295,a -104.7341,b 4.24502897,c -178.286896,s 2,t 11,e1 0.0,e2 0.0,e3 0.0,e4 0.0,e5 0.0,e6 0.0}
DECL FDAT FP766={TOOL_NO 1,BASE_NO 0,IPO_FRAME #BASE}
DECL LDAT LCPDAT222={VEL 2.0,ACC 100.0,APO_DIST 100.0,APO_FAC 50.0}
DECL E6POS XP767={x 1026.93103,y 887.223511,z 1172.96497,a -104.7342,b 4.2455368,c -178.286606,s 2,t 11,e1 0.0,e2 0.0,e3 0.0,e4 0.0,e5 0.0,e6 0.0}
DECL FDAT FP767={TOOL_NO 1,BASE_NO 0,IPO_FRAME #BASE}
DECL LDAT LCPDAT223={VEL 2.0,ACC 100.0,APO_DIST 100.0,APO_FAC 50.0}
DECL E6POS XP768={x 950.797424,y 809.914124,z 1172.96301,a -104.733597,b 4.24512291,c -178.286606,s 2,t 11,e1 0.0,e2 0.0,e3 0.0,e4 0.0,e5 0.0,e6 0.0}
DECL FDAT FP768={TOOL_NO 1,BASE_NO 0,IPO_FRAME #BASE}
DECL LDAT LCPDAT224={VEL 2.0,ACC 100.0,APO_DIST 100.0,APO_FAC 50.0}
DECL E6POS XP769={x 950.798401,y 809.911926,z 1282.15601,a -104.734001,b 4.2453208,c -178.286499,s 2,t 11,e1 0.0,e2 0.0,e3 0.0,e4 0.0,e5 0.0,e6 0.0}
DECL FDAT FP769={TOOL_NO 1,BASE_NO 0,IPO_FRAME #BASE}
